0: (*Einschwingvorgang wird abgewartet*)
	BereitNachstePosition:= FALSE;
	IF ManuellOK THEN 
	timer_Einschwingen(IN:= TRUE, PT:= T#120S ); // der Timer wird gestartet, damit sich das Wägesystem einschwingen kann
	IF timer_Einschwingen.Q  THEN 
		timer_Einschwingen(IN :=FALSE); 
		ManuellOK := FALSE;
		state:=1;
	END_IF
	END_IF
	
1: (*Kalibrierungsdaten werden aufgenommen und über einen FIlter gemittelt*)
	
	timer_Messen(IN:= TRUE, PT:= T#120S); //120 Sekunden wird gemessen
	
	CASE  Kalibrierungsschritt OF
		1: 
			GesKaliGewicht := Kalibrierungsgewichte[1];
			//SM.Mitteilung  :='Bitte hängen';
		2:
			GesKaliGewicht := Kalibrierungsgewichte[2];
		3:
			GesKaliGewicht := Kalibrierungsgewichte[1] + Kalibrierungsgewichte [2];
		4:
			GesKaliGewicht := Kalibrierungsgewichte[2] + Kalibrierungsgewichte [3];
		5:
			GesKaliGewicht := Kalibrierungsgewichte[1] + Kalibrierungsgewichte [2]+ Kalibrierungsgewichte [3];
	END_CASE

	FilterIn :=Waage_Offset[WaagenNummer]/ GesKaliGewicht;
	Trigger(in:= FilterIn, PT:= T#1S, out=> , Trig=> );

	WertMitteln(IN:= Trigger.out, E:= Trigger.Trig, N:= 30, RST:= BereitNachstePosition, AVG=>k_werte[Kalibrierungsschritt] );	
	
	IF timer_Messen.Q THEN 
		state :=2;
		timer_Messen(IN:= FALSE);
	END_IF


2: (*Übertragung der k-Werte in das Kalibrierungs-Array*)

	Umrechnungsfaktoren[WaagenNummer,Kalibrierungsschritt]:= k_werte[Kalibrierungsschritt];

	state:= 3;

3:	

	BereitNachstePosition:= TRUE;
	Kalibrierungsschritt:= Kalibrierungsschritt + 1; //nächster Kalibrierungsschritt
	
	(*Falls eine Waage alle Kalibrierungsschritte durchlaufen hat wird die nächste Waage 
		kalibriert.*)
	IF Kalibrierungsschritt > 5 THEN 
		WaageKalibriert[WaagenNummer]:=TRUE;
		WaagenNummer := WaagenNummer +1 ;
		Kalibrierungsschritt := 1;
		state:= 0;
	END_IF
	
	(*Alle Waagen sind alle 5 Kalibrierungsschritte durchlaufen. Gewichtskalibrierung ist abgeschlossen
		state wird auf Null gesetzt.*)
	IF Kalibrierungsschritt > 5  AND WaagenNummer > 4 THEN 
			WaagenKalibrierungFertig:= TRUE; 
			state:= 0;
	END_IF

END_CASE

END_PROGRAM

// ---- POUs/Waagen/Lesen_Waagen.TcPOU
PROGRAM Lesen_Waagen
(* Dieses Program wird dazu verwendet den aktuellen Waagenwert(String) aus dem Zwischenspeicher (RxBuffer) 
	zu entnehmen. Nach der Verarbeitung im Funktionsbaustein werden alle Werte der Waage_X wieder sich
	zugewiesen und gespeichert. *)  

VAR
	fb_WaageAuslesen : ARRAY[1..6] OF FB_GewichtAuslesen;
	counter: INT;
	myOffset: REAL;
	
(*Variablen für Offset-Ermittlung *)
	Timer,Timer1: TON;
	Trigger:  ARRAY[1..4] OF SH_1;
	GetOffset:ARRAY[1..4] OF FT_AVG;;
	bOffset: 		BOOL := FALSE;
	//bGetOffset: 		BOOL;

	Offset_VD: BOOL;
END_VAR

VAR PERSISTENT 
	Offset_Tare: 	ARRAY[1..4] OF REAL; 
	Offset_Ventilator_AN: 		ARRAY[1..4] OF REAL; 
	Offset_Kaltemittel_g: 		ARRAY[1..4] OF REAL; 
	Offset_Kaltemittel_f: 		ARRAY[1..4] OF REAL; 
END_VAR

// 	Waagen 1..6 werden ausgelesen. 
FOR counter:= 1 TO 6 DO 
	fb_WaageAuslesen[counter](myWaage:= Waage[counter] , myBuffer:= RxBuffer[counter] , Waage=> Waage[counter] );
	Waage_roh[counter] := Waage[counter].Masse;
END_FOR

(*Offset für Ventilator wird immer berücksichtig, wenn VD an ist und keine Kalibrierung geschieht*)
IF DO_VD_Ventilator_ON= TRUE AND bGetOffset_Ventilator = FALSE THEN
	Offset_VD := TRUE;
	ELSE
	Offset_VD := FALSE;
END_IF


(*	Waagen 1..4 werden falls nötig mit einem OFFSET korrigiert. zB durch Laufen der Ventilatoren.
 OFFSET wird nicht berechnet, wenn der gerade ein Offset ermittelt wird*)

IF 	bTare = FALSE 	THEN
//AND bGetOffset_Ventilator = FALSE AND bGetOffset_Kaltemittel_g = FALSE AND	bGetOffset_Kaltemittel_l = FALSE THEN
FOR counter:= 1 TO 4 DO 
	Waage_Offset[counter] := OFFSET(
	X:= Waage[counter].Masse, 
	O1:= bOffset, 				//wird TRUE nach dem ersten TARE-Befehl. Waagen sind wieder bei '0g'
	O2:= Offset_VD, 
	O3:= VD_Kaltemittel_g, 
	O4:= VD_Kaltemittel_l, 
	D:=  FALSE, 
	Offset_1:= -Offset_Tare[counter],
	Offset_2:= -Offset_Ventilator_AN[counter],  
	Offset_3:= -Offset_Kaltemittel_g[counter], 
	Offset_4:= -Offset_Kaltemittel_f[counter], 
	default:= 10000);
END_FOR
END_IF



//CASE SM.Status OF
	
//Initialisieren: 

IF 	bTare 	OR bGetOffset_Ventilator 	 OR bGetOffset_Kaltemittel_g OR	bGetOffset_Kaltemittel_l THEN 
	bGetOffset_Abgeschlossen	:=FALSE;
	bTare_Abgeschlossen 		:=FALSE;
	bVentilator_Abgeschlossen	:=FALSE;
	Timer(IN:= TRUE, PT:=T#60S , Q=> , ET=> );
	bOffset 					:= TRUE;
	IF bTare THEN 
		bOffset:= FALSE;
	END_IF
END_IF

//Offset wird bestimmt für den Fall, dass die Waagen mit ca. 2000 g vorbelastet sind
	IF bTare THEN 
		FOR counter:= 1 TO 4 DO 
			Trigger[counter](in:= Waage[counter].Masse, PT:= T#1S, out=> , Trig=> );
			GetOffset[counter](IN:= Trigger[counter].out, E:= Trigger[counter].Trig, N:= 30, RST:= , AVG=>Offset_Tare[counter] );	
		END_FOR
			//bOffset:= TRUE;
	END_IF


//Offset wird bestimmt für den Fall, dass der VENTILATOR an ist
	IF bGetOffset_Ventilator THEN
		VD_Ventilator_ON:= TRUE;
		Timer1(IN:=TRUE, PT:= T#30S); 
		IF Timer1.Q THEN 
			FOR counter:= 1 TO 4 DO 
				Trigger[counter](in:= Waage_Offset[counter], PT:= T#1S, out=> , Trig=> );//Trigger[counter](in:= Waage[counter].Masse, PT:= T#1S, out=> , Trig=> );
				GetOffset[counter](IN:= Trigger[counter].out, E:= Trigger[counter].Trig, N:= 30, RST:= , AVG=>Offset_Ventilator_AN[counter] );	
			END_FOR
		//Timer1(IN:=FALSE);
		END_IF
	END_IF

//Offset wird bestimmt für den Fall, dass das KÄLTEMITTEL GASFÖRMIG ist
	IF bGetOffset_Kaltemittel_g THEN 
		FOR counter:= 1 TO 4 DO 
			Trigger[counter](in:= Waage[counter].Masse, PT:= T#1S, out=> , Trig=> );
			GetOffset[counter](IN:= Trigger[counter].out, E:= Trigger[counter].Trig, N:= 30, RST:= , AVG=>Offset_Kaltemittel_g[counter] );	
		END_FOR
	END_IF

//Offset wird bestimmt für den Fall, dass das KÄLTEMITTEL FLÜSSIG ist	
	IF bGetOffset_Kaltemittel_l THEN 	
		FOR counter:= 1 TO 4 DO 
			Trigger[counter](in:= Waage[counter].Masse, PT:= T#1S, out=> , Trig=> );
			GetOffset[counter](IN:= Trigger[counter].out, E:= Trigger[counter].Trig, N:= 30, RST:= , AVG=>Offset_Kaltemittel_f[counter] );	
		END_FOR
	END_IF

//Nachdem die Zeit abgelaufen ist, werden die BOOL-Variablen zurückgesetzt
	IF Timer.Q THEN
		
		//bOffset								:= TRUE;
		
		bGetOffset_Kaltemittel_g			:= FALSE; 
		bGetOffset_Kaltemittel_l 			:= FALSE;
	
		IF bGetOffset_Ventilator = TRUE THEN
			VD_Ventilator_ON	:=		FALSE;
			bGetOffset_Ventilator:=		FALSE;
			bVentilator_Abgeschlossen:=	TRUE;
		END_IF
	
		IF bTare= TRUE THEN 
			bOffset						:= TRUE; //ermittelter Offset wird wieder vom Rohwert abgezogen
			bGetOffset_Abgeschlossen	:= TRUE;	
			bTare    					:= FALSE;
		END_IF
		Timer(IN:= FALSE);	
		Timer1(IN:=FALSE);
	END_IF
	
//END_CASE

END_PROGRAM

// ---- POUs/Funktionen/FB_GewichtAuslesen.TcPOU
FUNCTION_BLOCK FB_GewichtAuslesen

VAR_INPUT
	myWaage: WAAGE_VAR;		// Eine Inputvariable myWaage wird als WAAGE_VAR deklariert.
END_VAR

VAR_IN_OUT
	myBuffer:ComBuffer;		// Ein Zwischenspeicher wird deklariert. Buffer immer als VAR_IN_OUT deklarieren
END_VAR

VAR

(*Es folgen Variabeln die der FB ReceiveString benötigt*)
	ReceiveString_Buffer:	ReceiveString;
	tTimeout: 				TIME;
	bReset: 				BOOL;
	bStringReceived:		BOOL;
	bbusy:					BOOL;
	bRxTimeout: 			BOOL;
	eError: 				ComError_t;
	stLastStringReceived: 	STRING;
	stReceivedString: 		STRING;


	Var1: INT;				//1.Stringlänge
	Var2: INT;				//2.Stringlänge
	Var3: INT;				//3.Stringlänge
	MyString: STRING(80);	//
	Position_g: INT;		// Position des Grammzeichens 'g'. Ausgabe von Waage nur bei stabilen Werten
END_VAR
VAR_OUTPUT
	Waage: WAAGE_VAR (*:= myWaage*) ;  
END_VAR

//Empfange Datenstring aus dem Datenpuffer RxBuffer der jeweiligen Waage
ReceiveString_Buffer(
	Prefix:= '', 
	Suffix:= '$R$N', 
	Timeout:=tTimeout , 
	Reset:=bReset , 
	StringReceived=>bStringReceived , 
	Busy=>bbusy , 
	Error=>eError, 
	RxTimeout=> bRxTimeout ,
	ReceivedString:= stReceivedString, 
	RXbuffer:= myBuffer);

//Übergabe des empfangenen Strings an MyString und Längenabfrage
MyString:= stReceivedString;
Var1:= LEN (MyString);


//Löschen von $R$N aus MyString und Längenabfrage
MyString := DELETE (MyString,4,16); 
Var2:= LEN (MyString);


//Löschen der Leerzeichen aus MyString und Längenabfrage
WHILE FIND(MyString,' ') <> 0 DO
	MyString:=DELETE (MyString,1,FIND(MyString,' '));
END_WHILE
Var3:= LEN (MyString);


(*Überprüfen ob ein stabiler Messwert an der Waage anliegt
	Falls 'g' in MySting vorhanden 		-> Boolvariable bStabilerWert TRUE
	Falls kein 'g' in MyString vorhanden-> Boolvariable bStabilerWert FALSE	*)
Position_g := FIND(MyString,'g');
CASE Position_g OF
		0: myWaage.bStabilerWert := FALSE;
	ELSE
		myWaage.bStabilerWert := TRUE;
END_CASE


// Übergabe von MyString in Realvariable MyReal

myWaage.Masse:=STRING_TO_REAL(MyString);

Waage:= myWaage;

END_FUNCTION_BLOCK

// ---- POUs/Modbus/Lesen_Modbus.TcPOU
PROGRAM Lesen_Modbus
(*In diesem Programm werden alle Modbus-Daten umgerechnet. *)

VAR
	Auslesen0, Auslesen1, Auslesen2, Auslesen3, Auslesen4, Auslesen5, Auslesen6, Auslesen7, Auslesen8 : FB_fpconverter;
	
	EV1 : FB_EVconverter;		//Funktionsbaustein zur Auswertung eines Expansionsventiles
	EV2 : FB_EVconverter;		//Funktionsbaustein zur Auswertung eines Expansionsventiles
	FP_Umrechnen : FB_fpconverter;	//Funktionsbaustein zur Umrechnung von FLOAT->REAL
END_VAR

(*Auslesen der Druckdaten der 8 Drucksensoren im Kältekreis*)
Auslesen1(myPT:= PT_KP_in, 	PT=> PT_KP_in);
Auslesen2(myPT:= PT_KP_out, PT=> PT_KP_out);
Auslesen3(myPT:= PT_VF_in,	PT=> PT_VF_in);
Auslesen4(myPT:= PT_VF_out, PT=>PT_VF_out );
Auslesen5(myPT:= PT_vor_EV, PT=>PT_vor_EV );
Auslesen6(myPT:= PT_vor_EV_rev, PT=>PT_vor_EV_rev );
Auslesen7(myPT:= PT_VD_in,  PT=> PT_VD_in);
Auslesen8(myPT:= PT_VD_out, PT=> PT_VD_out);

(*Deklarierung der ModbusData_Startfelder der Slaves Modbus. Hier schreibt der ModbusRTU die empfangenden Daten hinein
	Startfeld entspricht zur Übersicht der Modbus-Adresse. *)
PT_KP_in.Startfeld_ModbusData		:= 4;
PT_KP_out.Startfeld_ModbusData		:= 5;
PT_VF_in.Startfeld_ModbusData		:= 6;
PT_VF_out.Startfeld_ModbusData		:= 7;
PT_vor_EV.Startfeld_ModbusData		:= 8;
PT_vor_EV_rev.Startfeld_ModbusData 	:= 9;
PT_VD_in.Startfeld_ModbusData		:= 10;
PT_VD_out.Startfeld_ModbusData		:= 11;

(*Expansionsventile werden ausgelesen und umgerechnet*)
EV1(inEV:=EV , outEV=> EV);
EV2(inEV:=EV_rev, outEV=> EV_rev);

(*Daten vom Massestromsensoren werden umgerechnet. FLOAT-Werte werden in REAL umgerechnet*)
MSS.rFliessgeschwindigkeit	:= FloatPointDW_TO_REAL(MSS.Data[1]);
MSS.rVolumenstrom			:= FloatPointDW_TO_REAL(MSS.Data[2]);
MSS.rMassenstrom			:= FloatPointDW_TO_REAL(MSS.Data[3])*1000; // wird nun angezeigt in [g/s]
MSS.rTemp					:= K_TO_C(FloatPointDW_TO_REAL(MSS.Data[4]));
MSS.rDichte					:= FloatPointDW_TO_REAL(MSS.Data[5]);

END_PROGRAM

// ---- POUs/Funktionen/FB_fpconverter.TcPOU
FUNCTION_BLOCK FB_fpconverter 
(* Dieser FB dient zur Umrechnung der DATABYTEs in einen REAL-Wert.
	Je nach ausgeführtem Modbus-Befehl(nur Druck oder Temperatur, oder beides) werden
	unterschiedlich viele DATABYTEs von dem Drucksensor geschickt. 
	Die Boolvariablen zur Druck- und Temperaturabfrage müssen durch den User gesetzt werden.
	Der FB gibt den Druck und die Temperatur in REAL an die STRUCT Drucksensor zurück.*)

VAR_INPUT
	myPT : Drucksensor;
END_VAR
VAR
	myString_druck: STRING(32);
	myString_temp: STRING(32);
END_VAR

VAR_OUTPUT
		PT: Drucksensor;
END_VAR

//Umrechnung der BYTEs in Binär-STRINGs und zusammensetzen der 4 DATA-BYTEs zu einem 32 bit STRING
myPT.Data[0]:= ModbusRTU_COM.modbusData_PT[myPT.Startfeld_ModbusData];

	IF myPT.bDruckabfrage THEN
		myString_druck:=DWORD_TO_BINSTRING(ModbusRTU_COM.modbusData_PT[myPT.Startfeld_ModbusData]);
		myPT.rDruck:=BINSTRING_TO_REAL(myString_druck); 		// tatsächlicher Druck in Bar
	ELSE
		myPT.rDruck:=0;	
	END_IF
	
	
(*Umrechnung für Temperatur, falls bTemperaturabfrage gleich TRUE *)	
	IF myPT.bTemperaturabfrage  THEN
		myString_druck:=DWORD_TO_BINSTRING(ModbusRTU_COM.modbusData_PT[myPT.Startfeld_ModbusData]);
		myPT.rTemp:= BINSTRING_TO_REAL(myBinString:= myString_temp); 		//Umrechnung nach IEEE 754 von 32 bit floating point zur REAL-Variable 
	ELSE
		myPT.rTemp:= 0;
	END_IF

PT := myPT;

END_FUNCTION_BLOCK

// ---- POUs/Modbus/ModbusRTU_COM.TcPOU
PROGRAM ModbusRTU_COM

(*Dieses Programm komuniziert über einen MODBUS-RTU mit den installieren Drucksensoren(PT),
den E-Ventilen und dem Massenstromsensor im Kältekreislauf. Die Senoren/Aktoren besitzen eine 
eindeutige Adresse. Über die Adressen werden sie vom MASTER(Pc) angesprochen und führen die
verlange Funktion durch.

Dieses Programm ist erst nach Initialierung, sprich Zuweisung der Adressen, zu verwenden.
Wenn mehrere Sensoren/Aktoren die gleiche Adresse haben, kommt es zu Fehlern in der Kommunikation.
Die Kommunikation verläuft in einer CASE-Struktur.*)

VAR
(*
_________________________________________________________	
Drucksensoren	|	Position im RI	|	Modbus-Adresse
PT_KP_in		|	1				|	4
PT_KP_out		|	2				|	5
PT_VF_in		|	2‘ 				|	6
PT_VF_out		|	3‘ 				|	7
PT_vor_EV 		|	3 (innerhalb KK)|	8 
PT_vor_EV_rev 	|	3 (außerhalb KK)|	9
PT_VD_in		|	4				|	10
PT_VD_out		|	1‘ 				|	11
__________________________________________________________
Massenstromsensor
MSS 1			|	3				|	12 
*)
	
	state: INT;

(*Variablen für die Modbus-Befehle*)
	 ModbusAdresse: 	BYTE := 3;
	 modbusData_PT: 	ARRAY[0..12] OF DWORD;		//hier werden die Daten von den Drucksensoren gespeichert
	 
(*Abfrageregister vom MassenstromSensor*)
	AbfrageRegs_MSS:ARRAY[1..5] OF INT := [30000,30002,30004,30006,30008]; 	

(*Abfrageregister vom MassenstromSensor*)
	AbfrageRegs_PT:WORD := 2; 	
	LaengeRegs: BYTE:= 2;
	
(*Variablen für Error- und Successzähler der Modbus-Komunikation *)
	FtrigBusy:			F_TRIG;
	LastErrorstate: 	INT;
	LastModbusError: 	ST_ModbusErrorDiagnostics;
	CounterError: 		DINT;
	CounterSuccess: 	DINT;
	counter: 			INT := 1;
	Teststring: T_MaxString;
END_VAR

(*Falls ein Slave konfiguriert werden soll bConfigPT auf TRUE setzen*)
		
IF 	bConfigPT THEN 
	Status_Modbus := ConfigPT;
ELSE 
	Status_Modbus := Aktiv;
END_IF


CASE Status_Modbus OF
	
Aktiv: 

CASE state OF

0: (*Initialisierung von Modbus und Durchzählen der Modbus-Adressen*)
		MODBUS.myModbus.ReadRegs(Execute:= FALSE);
		MODBUS.myModbus.WriteRegs(Execute:= FALSE);

		
		ModbusAdresse := ModbusAdresse + 1;		//Laufvariable für die ModbusAdressen der Slaves. Zunächst nur Drucksensoren.
		IF ModbusAdresse >= 13 THEN				//alle PTs und der Massenstromsensor werden ausgelesen
			ModbusAdresse := 4;
		END_IF
		
		
		state := state + 1;


1:	(* Lese Keller-Registers aus*)	
     
	IF ModbusAdresse<=11 AND ModbusAdresse>=4 THEN 
	 MODBUS.myModbus.ReadRegs (* Reads data from a connected slave. *)
 		(
 		 UnitID:= ModbusAdresse,
 		 Quantity:= LaengeRegs,								//zwei Register werden ausgelesen
 		 MBAddr:= AbfrageRegs_PT,								//P1 wird bei Adresse 2 ausgelesen, TOB1 bei Adresse 8
 		 cbLength:= SIZEOF(modbusData_PT[ModbusAdresse]),		
 		 pMemoryAddr:= ADR(modbusData_PT[ModbusAdresse]),		//Empfangene Daten werden in DWORD in modbusData geschrieben.
  		Execute:= TRUE,
  		Timeout:= modbusTimeout,
  		Busy => Modbus.isModbusBusy,
  		Error => isModbusError,
  		ErrorId => modbusErrorId
  		(* cbRead parameter *));
		
  		IF NOT isModbusBusy THEN
				MODBUS.myModbus.ReadRegs(Execute:= FALSE);
			IF MODBUS.myModbus.Error THEN
				state := 0;
			ELSE
				state := state + 1;
			END_IF
		END_IF
		ELSE 
		state := state + 1;
	END_IF
	
	
	
2:	(* Lese Massenstromsensor-Registers aus*)		
	(*	Folgende Messdaten werden ausgelesen:
			
				   Messgröße		|	Einheit	|	Register-Adressen
				____________________|___________|_____________________   
				1) Fließgeschw.     |	[m/s]	|	30000-2 Regs
				2) Volumenstrom		|	[m³/s]	|	30002-2 Regs
				3) Massenstrom		|	[kg/s]	|	30004-2 Regs
				4) Temperatur		|	[K]		|	30006-2 Regs
				5) Dichte			|	[kg/m³]	|	30008-2 Regs			->ingesamt 10 Regs
		*) 
	IF ModbusAdresse=12 THEN	
		myModbus.ReadInputRegs(
		UnitID:= 12,
 		Quantity:= 2,							
 		MBAddr:= INT_TO_WORD(AbfrageRegs_MSS[counter]),								
 		cbLength:= SIZEOF(MSS.Data[counter]),		
 		pMemoryAddr:= ADR(MSS.Data[counter]),	 
  		Execute:= TRUE,
  		Timeout:= modbusTimeout,
  		Busy => isModbusBusy,
  		Error => isModbusError,
  		ErrorId => modbusErrorId
  		(*cbRead parameter)*));
	
			IF isModbusBusy = FALSE AND counter<=5 THEN
				myModbus.ReadInputRegs(Execute:= FALSE);
				counter:= counter +1;
			END_IF	
			
			IF isModbusBusy = FALSE AND counter>5 THEN
				myModbus.ReadInputRegs(Execute:= FALSE);
				counter:=1;
				state:= 0;
			END_IF	
	ELSE 
		state:= 0;
	END_IF	
END_CASE	

ConfigPT:
	
	ConfigDrucksensor(); 		//Programm für Konfigurierung von Keller-Drucksensoren

END_CASE 

// Zählen der erfolgreichen und fehlerhaften Komunikationsschritte 
FtrigBusy(CLK:=myModbus.BUSY );
IF FtrigBusy.Q THEN
	IF MODBUS.myModbus.Error THEN
		LastModbusError := MODBUS.myModbus.ErrorDiagnostics;
		LastErrorstate := state;
		CounterError := CounterError + 1;
	ELSE
		CounterSuccess := CounterSuccess + 1;
	END_IF
END_IF

END_PROGRAM

// ---- POUs/Modbus/ConfigDrucksensor.TcPOU
PROGRAM ConfigDrucksensor
VAR
	state : INT := 1;
	
	(*Daten für die Konfiguration vom Keller-Drucksensor*)	
	UART_akt: 				WORD;
	UARTsettings_akt:		ARRAY[0..1]OF BYTE;
	UARTsettings_neu: 		ARRAY[0..1]OF BYTE  ;//:= [48,0];
	wUARTsettings_neu:		WORD := 0;//:= 112;
	sUARTsettings_neu: 		STRING;
	ModbusRegister:   		Word := 17;
	RegisterLange: 			BYTE := 1;
	ModbusAddress_alt: 		WORD {1..250}:= 1;			//alte Modbusadresse des Slaves. Anfangs gleich der Auslieferungsadresse
	ModbusAddress_neu: 		WORD {3..12} := 11;				//neue Modbusadresse des Slaves. 
	ModbusDataTest: 		DWORD;
	Teststring: 			STRING;
END_VAR

(*Keller-Slaves Konfiguration*)

Teststring:= DWORD_TO_BINSTR(ModbusDataTest,32);

CASE MODBUS.Status_Modbus OF

ConfigPT:

CASE state OF
1:   (* Write Register, write new address to Slave *)	
		IF bConfigPT_setadresse THEN
	 	MODBUS.myModbus.WriteSingleRegister (* writes data to a connected slave. *)
 		(
 		 UnitID:= WORD_TO_BYTE(ModbusAddress_alt),
 		 Quantity:= 1,
 		 MBAddr:= 525,							//Keller: DEV_ADDR 0x020D= DECx525
 		 cbLength:= SIZEOF(ModbusAddress_neu),
 		 pMemoryAddr:= ADR(ModbusAddress_neu),
  		Execute:= TRUE,
  		Timeout:= modbusTimeout,
  		Busy => isModbusBusy,
  		Error => isModbusError,
  		ErrorId => modbusErrorId
  		(* cbRead parameter *));
		
  		IF NOT isModbusBusy THEN
				MODBUS.myModbus.WriteSingleRegister(Execute:= FALSE);
			IF MODBUS.myModbus.Error THEN
				state := 2;
			ELSE
				state := 2;	
			END_IF
		END_IF
		ELSE
			state:= 2;
		END_IF
	
2: 	(* TEST-READ Regs from connected Slave *)

		 MODBUS.myModbus.ReadRegs 
 		(
 		 UnitID:= WORD_TO_BYTE(ModbusAddress_neu),
 		 Quantity:= RegisterLange,						//2 Regs für den Druck P1 oder Temperatur TOB1
 		 MBAddr:= ModbusRegister,						//DECx02 Reg-Adresse für P1, DECx08 Reg-Adresse für TOB1
 		 cbLength:= SIZEOF(ModbusDataTest),
 		 pMemoryAddr:= ADR(ModbusDataTest),
  		Execute:= TRUE,
  		Timeout:= modbusTimeout,
  		Busy => isModbusBusy,
  		Error => isModbusError,
  		ErrorId => modbusErrorId
  		(* cbRead parameter *));
		
  		IF NOT isModbusBusy THEN
				MODBUS.myModbus.ReadRegs(Execute:= FALSE);
			IF myModbus.Error THEN
				state := 2;
			ELSE
				state := 1;	
			END_IF
		END_IF
		
3: (* Write Register, write new UART-settings to Slave *)
	IF bConfigPT_setUART THEN
	 	MODBUS.myModbus.WriteSingleRegister (* writes data to a connected slave. *)
 		(
 		 UnitID:= WORD_TO_BYTE(ModbusAddress_neu),
 		 Quantity:= 1,
 		 MBAddr:= 512,							//Keller: DEV_ADDR 0x020D= DECx525
 		 cbLength:= SIZEOF(wUARTsettings_neu),
 		 pMemoryAddr:= ADR(wUARTsettings_neu),
  		Execute:= TRUE,
  		Timeout:= modbusTimeout,
  		Busy => isModbusBusy,
  		Error => isModbusError,
  		ErrorId => modbusErrorId
  		(* cbRead parameter *));
		
		sUARTsettings_neu:= CONCAT(BYTE_TO_STRING(UARTsettings_neu[1]), BYTE_TO_STRING(UARTsettings_neu[0]));
  		IF NOT isModbusBusy THEN
				MODBUS.myModbus.WriteSingleRegister(Execute:= FALSE);
			IF MODBUS.myModbus.Error THEN
				state := 1;
			ELSE
				state := 4;	
			END_IF
		END_IF
	ELSE
		state:= 4;
  	END_IF

4: (* Read UART-Register from Slave *)

	 	MODBUS.myModbus.ReadRegs
 		(
 		 UnitID:= WORD_TO_BYTE(ModbusAddress_neu),
 		 Quantity:= 1,
 		 MBAddr:= 512,							//Keller: DEV_ADDR 0x020D= DECx525
 		 cbLength:= SIZEOF(UARTsettings_akt),
 		 pMemoryAddr:= ADR(UARTsettings_akt),
  		Execute:= TRUE,
  		Timeout:= modbusTimeout,
  		Busy => isModbusBusy,
  		Error => isModbusError,
  		ErrorId => modbusErrorId
  		(* cbRead parameter *));
		
		//Ändert die Byte-Reihenfolge und konvertiert sie in ein WORT
		UART_akt:= WORD_OF_BYTE(UARTsettings_akt[1], UARTsettings_akt[0]);
		
		
  		IF NOT isModbusBusy THEN
				MODBUS.myModbus.ReadRegs(Execute:= FALSE);
			IF MODBUS.myModbus.Error THEN
				state := 3;
			ELSE
				state := 4;	
			END_IF
		END_IF
		
END_CASE

END_CASE

END_PROGRAM

// ---- POUs/Funktionen/DWORD_TO_BINSTRING.TcPOU
FUNCTION DWORD_TO_BINSTRING : STRING(32)
VAR_INPUT
	myDWORD:DWORD;		//DWORD aus der Klemme/Modbusarray
END_VAR
VAR
		b3: BYTE; 
		b2: BYTE;
		b1: BYTE;
		b0: BYTE;
		s3: STRING(8);
		s2: STRING(8);
		s1: STRING(8);
		s0: STRING(8);
END_VAR

(*da Twincat mit LIL-Endian arbeitet und die Kellersensoren mit BIG-Endian,
 müssen die Bytes paarweise vertauscht werden*)

//Zerteilen des DWORDs in die 4 Bytes
b3:= BYTE_OF_DWORD(myDWORD, 1);
b2:= BYTE_OF_DWORD(myDWORD, 0);
b1:= BYTE_OF_DWORD(myDWORD, 3);
b0:= BYTE_OF_DWORD(myDWORD, 2);

//Umrechnung der BYTES in Binärestrings mit der Länge 8 bits
s3:= BYTE_TO_BINSTR(b3,8);
s2:= BYTE_TO_BINSTR(b2,8);
s1:= BYTE_TO_BINSTR(b1,8);
s0:= BYTE_TO_BINSTR(b0,8);

//Zusammenfügen der vier Binärstrings zu einem 32 bit String
DWORD_TO_BINSTRING := CONCAT(CONCAT(s3,s2), CONCAT(s1,s0));

END_FUNCTION

// ---- POUs/Funktionen/BINSTRING_TO_REAL.TcPOU
FUNCTION BINSTRING_TO_REAL : REAL
	(*Ein 32 bit Binärstring wird in einen REAL-Wert umgerechnet*)
VAR_INPUT
	myBinString : STRING(32);
END_VAR
VAR
	stSign: STRING(1);
	rSign: 	REAL;
	Sign: 	BOOL;
	
	stExponent: STRING(8);
	Exponent: 	UINT;
	
	stMantis: 	STRING(23);
	Mantis: 	DWORD;

END_VAR

	
	stSign		:= LEFT(myBinString,1);
	Sign		:= STRING_TO_BOOL(stSign);
	rSign		:= STRING_TO_REAL(stSign);

	stExponent	:= RIGHT(LEFT(myBinString,9),8);	
	Exponent	:= BYTE_TO_UINT(BIN_TO_BYTE(stExponent));

	stMantis	:= RIGHT(myBinString,23);
	Mantis		:= BIN_TO_DWORD(stMantis);

	BINSTRING_TO_REAL:= FPU.ComposeRealRaw(bS:=Sign , uiE:= Exponent, udiM:= Mantis ); // Ergebnis in REAL

END_FUNCTION

// ---- POUs/Funktionen/FB_EVconverter.TcPOU
FUNCTION_BLOCK FB_EVconverter
VAR_INPUT
	inEV : ExpansionsVentil;
END_VAR
VAR
END_VAR

VAR_OUTPUT
	 outEV : ExpansionsVentil;
END_VAR

	inEV.IstDruck :=	 	INT_TO_REAL(WORD_TO_INT(inEV.modbusData[1]))/10;
	inEV.IstTemp:=	 		INT_TO_REAL(WORD_TO_INT(inEV.modbusData[2]))/10;
	inEV.SaugTemp:= 		INT_TO_REAL(WORD_TO_INT(inEV.modbusData[3]))/10;
	inEV.VerdampfTemp:= 	INT_TO_REAL(WORD_TO_INT(inEV.modbusData[4]))/10;
	inEV.VerdampfDruck:= 	INT_TO_REAL(WORD_TO_INT(inEV.modbusData[5]))/10;
	inEV.UberhitzungTemp:= 	INT_TO_REAL(WORD_TO_INT(inEV.modbusData[6]))/10;
	inEV.VentilOffnung:= 	INT_TO_REAL(WORD_TO_INT(inEV.modbusData[7]))/10;
	inEV.RegelSollwert:= 	INT_TO_REAL(WORD_TO_INT(inEV.modbusData[8]))/10;
	inEV.Ventilposition:= 	INT_TO_REAL(WORD_TO_INT(inEV.modbusData[9]));
	inEV.AktKuhlleistung:= 	INT_TO_REAL(WORD_TO_INT(inEV.modbusData[10]));
	
	inEV.LOP := inEV.modbusDataCoils[1];
	inEV.MOP := inEV.modbusDataCoils[2];
	inEV.LowSH:= inEV.modbusDataCoils[3];
	inEV.HiTcond:= inEV.modbusDataCoils[4];
	
	outEV:= inEV;

END_FUNCTION_BLOCK

// ---- POUs/Funktionen/FloatPointDW_TO_REAL.TcPOU
FUNCTION FloatPointDW_TO_REAL : REAL
(*Diese Funktions rechnet 32 bit FLOAT-Werte in einen REAL-Wert um und gibt diesen wieder aus.*)
VAR_INPUT
	in : DWORD;
END_VAR
VAR
	BinString : STRING;
END_VAR

(*DWORD wird in einen Binären 32bit String umgewandelt*) 
BinString:= DWORD_TO_BINSTR(in,32);
 
 (*Binärstring wird in eine REAL Variable umgerechnet*)
 FloatPointDW_TO_REAL:= BINSTRING_TO_REAL(myBinString:= BinString);

END_FUNCTION

// ---- POUs/Modbus/ModbusRTU_EL.TcPOU
PROGRAM ModbusRTU_EL
VAR
(*Modbus für Klemme EL6021 wird deklariert*)
	ModbusEL6021:		ModbusRtuMaster_KL6x22B;	
	modbusTimeout_EL:	TIME := T#300MS;
	isModbusBusy_EL:	BOOL;
	isModbusError_EL:	BOOL;
	modbusErrorId_EL:	MODBUS_ERRORS;
	
(*Hilfsvariablen für Modbus	

Sensor/Aktor	|	Position		|	Modbus-Adresse
________________|___________________|____________________
EV				|	3				|	2
EV_rev			|	3				|	3	
*)
	//modbusData_EV: 	ARRAY[1..10] OF INT;		//hier werden die Daten vom EV gespeichert
	EV_Adresse : BYTE := 2;				//ModbusAdresse vom Expansionsventil	
	EV_rev_Adresse : BYTE := 3;			//ModbusAdresse vom Abtau-Expansionsventil
	state: 			INT := 0;
	counter: 		INT := 1;
	
	AbfrageRegs: ARRAY [1..10] OF WORD := [0,1,4,5,6,9,16,20,131,134]; 	//Modbus-Register-Adressen. Das sind alle Werte die vom EV abgefragt werden
	AbfrageCoils: ARRAY [1..4] OF WORD := [49,50,51,52];					//Modbus-Coil-Adressen.
	
(*Variablen für Error- und Successzähler der Modbus-Komunikation *)
	FtrigBusy:			F_TRIG;
	LastErrorstate: 	INT;
	LastModbusError: 	ST_ModbusErrorDiagnostics;
	CounterError: 		DINT;
	CounterSuccess: 	DINT;

	TestMSS: ARRAY [0..10] OF DWORD;
END_VAR


CASE state OF

0: (*Initialisierung von Modbus*)
	
		ModbusEL6021.ReadInputRegs(Execute:= FALSE);
		ModbusEL6021.ReadCoils(Execute:= FALSE);
		ModbusEL6021.WriteSingleRegister(Execute:= FALSE);

		state :=1;
		
1: (*Liest Register von EV aus*)
 	
		ModbusEL6021.ReadInputRegs(
		UnitID:= EV_Adresse,
 		Quantity:= 1,								
 		MBAddr:= AbfrageRegs[counter],								
 		cbLength:= SIZEOF(EV.modbusData[counter]),//EV.modbusData[counter]),		
 		pMemoryAddr:= ADR(EV.modbusData[counter]),//EV.modbusData[counter]),		//Daten werden in für EV DATA-ARRAY geschrieben
  		Execute:= TRUE,
  		Timeout:= modbusTimeout_EL,
  		Busy => isModbusBusy_EL,
  		Error => isModbusError_EL,
  		ErrorId => modbusErrorId_EL
  		(*cbRead parameter)*));

		IF NOT isModbusBusy_EL THEN
				ModbusEL6021.ReadInputRegs(Execute:= FALSE);
			IF MODBUS.myModbus.Error THEN
				state := 0;
				ELSE
				counter := counter + 1;	
					IF counter > 10 THEN		//alle deklarierten Modbus-Register werden ausgelesen
					counter := 1;
					state:= 2;
					END_IF
			END_IF
		END_IF
		


	
2: (*Liest Coils von EV aus*)
		ModbusEL6021.ReadCoils(
		UnitID:= EV_Adresse,
 		Quantity:= 1,								
 		MBAddr:= AbfrageCoils[counter],								
 		cbLength:= SIZEOF(EV.modbusDataCoils[counter]),		
 		pMemoryAddr:= ADR(EV.modbusDataCoils[counter]),		//Daten werden in für EV DATA-ARRAY geschrieben
  		Execute:= TRUE,
  		Timeout:= modbusTimeout_EL,
  		Busy => isModbusBusy_EL,
  		Error => isModbusError_EL,
  		ErrorId => modbusErrorId_EL
  		(*cbRead parameter)*));
		
		IF NOT isModbusBusy_EL THEN
				ModbusEL6021.ReadCoils(Execute:= FALSE);
			IF ModbusEL6021.Error THEN
				state := 0;
			ELSE
				counter:= counter+1;
				IF counter > 4 THEN		//alle deklarierten Modbus-Register werden ausgelesen
					counter := 1;
					state:= 3;
				END_IF
			END_IF
		END_IF
		
3: (*Schreibt Akt_Kühlleistung Coil auf die Expansionsventile*)
IF EV.SetKuhlleistung THEN 	
	ModbusEL6021.WriteSingleRegister(
		UnitID:= EV_Adresse,
 		Quantity:= 1,								
 		MBAddr:= 134,								
 		cbLength:= SIZEOF(EV.SollKuhlleistung),		
 		pMemoryAddr:= ADR(EV.SollKuhlleistung),		//Daten werden in für EV DATA-ARRAY geschrieben
  		Execute:= TRUE,
  		Timeout:= modbusTimeout_EL,
  		Busy => isModbusBusy_EL,
  		Error => isModbusError_EL,
  		ErrorId => modbusErrorId_EL
  		(*cbRead parameter)*));

		IF NOT isModbusBusy_EL THEN
				ModbusEL6021.WriteSingleRegister(Execute:= FALSE);
				EV.SetKuhlleistung := FALSE;
			IF ModbusEL6021.Error THEN
				state := 0;
			ELSE
				state:= 4;
			END_IF
		END_IF
	ELSE 
		state:= 4;
END_IF
	
4: (*Liest Register von EV_rev aus*)
 	
		ModbusEL6021.ReadInputRegs(
		UnitID:= EV_rev_Adresse,
 		Quantity:= 1,								
 		MBAddr:= AbfrageRegs[counter],								
 		cbLength:= SIZEOF(EV_rev.modbusData[counter]),//EV.modbusData[counter]),		
 		pMemoryAddr:= ADR(EV_rev.modbusData[counter]),//EV.modbusData[counter]),		//Daten werden in für EV DATA-ARRAY geschrieben
  		Execute:= TRUE,
  		Timeout:= modbusTimeout_EL,
  		Busy => isModbusBusy_EL,
  		Error => isModbusError_EL,
  		ErrorId => modbusErrorId_EL
  		(*cbRead parameter)*));

		IF NOT isModbusBusy_EL THEN
				ModbusEL6021.ReadInputRegs(Execute:= FALSE);
			IF MODBUS.myModbus.Error THEN
				state := 0;
				ELSE
				counter := counter + 1;	
					IF counter > 10 THEN		//alle deklarierten Modbus-Register werden ausgelesen
					counter := 1;
					state:= 5;
					END_IF
			END_IF
		END_IF
		


	
5: (*Liest Coils von EV_rev aus*)
		

		ModbusEL6021.ReadCoils(
		UnitID:= EV_rev_Adresse,
 		Quantity:= 1,								
 		MBAddr:= AbfrageCoils[counter],								
 		cbLength:= SIZEOF(EV_rev.modbusDataCoils[counter]),		
 		pMemoryAddr:= ADR(EV_rev.modbusDataCoils[counter]),		//Daten werden in für EV DATA-ARRAY geschrieben
  		Execute:= TRUE,
  		Timeout:= modbusTimeout_EL,
  		Busy => isModbusBusy_EL,
  		Error => isModbusError_EL,
  		ErrorId => modbusErrorId_EL
  		(*cbRead parameter)*));

		IF NOT isModbusBusy_EL THEN
				ModbusEL6021.ReadCoils(Execute:= FALSE);
			IF ModbusEL6021.Error THEN
				state := 0;
			ELSE
				counter:= counter+1;
				IF counter > 4 THEN		//alle deklarierten Modbus-Register werden ausgelesen
					counter := 1;
					state:= 6;
				END_IF
			END_IF

		END_IF

6: (*Schreibt Akt_Kühlleistung Coil auf die Expansionsventile*)

IF EV_rev.SetKuhlleistung THEN 	
	ModbusEL6021.WriteSingleRegister(
		UnitID:= EV_rev_Adresse,
 		Quantity:= 1,								
 		MBAddr:= 134,								
 		cbLength:= SIZEOF(EV_rev.SollKuhlleistung),		
 		pMemoryAddr:= ADR(EV_rev.SollKuhlleistung),		//Daten werden in für EV DATA-ARRAY geschrieben
  		Execute:= TRUE,
  		Timeout:= modbusTimeout_EL,
  		Busy => isModbusBusy_EL,
  		Error => isModbusError_EL,
  		ErrorId => modbusErrorId_EL
  		(*cbRead parameter)*));

		IF NOT isModbusBusy_EL THEN
				ModbusEL6021.WriteSingleRegister(Execute:= FALSE);
				EV_rev.SetKuhlleistung := FALSE;
			IF ModbusEL6021.Error THEN
				state := 0;
			ELSE
				state:= 0;
			END_IF
		END_IF
	ELSE 
		state:= 0;
END_IF	
END_CASE

FtrigBusy(CLK:=ModbusEL6021.BUSY );
(*zählt fehlgeschlagene und erfolgreiche Komunikationsschritte*)
IF FtrigBusy.Q THEN
	IF ModbusEL6021.Error THEN
		LastModbusError := ModbusEL6021.ErrorDiagnostics;
		LastErrorstate := state;
		CounterError := CounterError + 1;
	ELSE
		CounterSuccess := CounterSuccess + 1;
	END_IF
END_IF

END_PROGRAM

// ---- POUs/Vereisung.TcPOU
PROGRAM Vereisung
(*Ablaufprogram für die Vereisung des Verdampfers. Beim ABBRUCH des Vorgangs bzw. ABSCHALTEN wird ein PumpDown vollzogen.  *)
VAR

END_VAR

(*Starte Timer zur Vereisung*)	
	IF NOT TimerVereisung.IN THEN
	TimerVereisung(IN:= TRUE, PT:= Vereisungszeit);
	END_IF
 		
	IF SM.bKuehlen THEN 
		fb_Schuetzstellung(myStatus := KuehlenOben);
	END_IF
	
(*Abtauung wird begonnen wenn Zeit des Timers abgelaufen ist*)
	IF TimerVereisung.Q THEN
		TimerVereisung.IN := FALSE;			//Reset vom Vereisungstimer
		Mitteilung:= 'Die Vereisungszeit ist abgeschlossen';
		
		(*Nach der Vereisung wird ein PumpDown durchgeführt*)
		SM.bPumpDown := TRUE; 
		
		(* Status-Maschine Bool-variablen werden auf TRUE bzw. FALSE gesetzt*)
		SM.bKuehlen := FALSE;	

		IF AutomatikZyklusEin THEN 
				bAbtauen := TRUE; 
				bPumpDown_revAbgeschlossen := FALSE;		//damit wieder ein PUMPDOWN rev im nächsten Zyklus durchgeführt werden kann
				CASE  AutomatikAbtauModus OF 
						NichtAusgewahlt: 
							Mitteilung := 'Kein Automatik-Abtaumodus ausgewählt!';
						Abtauen_elektrisch:
							bAbtauen_elektrisch := TRUE;
						Abtauen_Heissgas_oben:
							bAbtauen_Heissgas_oben:= TRUE;
						Abtauen_Heissgas_unten:
							bAbtauen_Heissgas_unten := TRUE;
				END_CASE
				
		END_IF	
	END_IF

END_PROGRAM

// ---- POUs/Funktionen/FB_Schuetzstellung.TcPOU
FUNCTION_BLOCK FB_Schuetzstellung
VAR_INPUT
myStatus: Status_Schuetzstellung;
END_VAR
VAR_OUTPUT
END_VAR
VAR
END_VAR

CASE  myStatus OF

KuehlenOben:
	(*Schütze werden geschaltet*)
		Schuetz_1K3 := TRUE;
		Schuetz_1K4 := FALSE;
		Schuetz_1K5 := TRUE;

	(*Falls Komponente ON ist wird sie auf TRUE gesetzt*)	
		VD_Ventilator_ON			:= TRUE; 
		VD_defrost_Ventilator_ON	:= FALSE;
		ElektrischeHeizung_ON		:= FALSE; 
		KP_ON						:= TRUE;  
		
	(*Expansionsventil wird aktiviert und auf 100% gestellt. Komunikation erfolgt über Modbus_EL*)
	IF  EV.SollKuhlleistung<> 100 THEN 
		EV.SetKuhlleistung := TRUE;
		EV.SollKuhlleistung:= 100;
	END_IF
	
	(*Expansionsventil für die Abtauung wird auf 100% zurückgestellt. Kann verändert werden, um Kälteleistung bzw. Abtaleistung zu variieren*)	
	IF EV_rev.SollKuhlleistung <> 100 THEN 
		EV_rev.SetKuhlleistung := TRUE;
		EV_rev.SollKuhlleistung:= 100;
	END_IF
	
PumpDown: (*Pump-Down wird durchgeführt bis der Druck vor dem KP kleiner als 1,4 Bar ist*)	
	
	(*Schütze werden geschaltet*)
		Schuetz_1K3 := TRUE;
		Schuetz_1K4 := FALSE;
		Schuetz_1K5 := TRUE;
		
	(*Falls Komponente ON ist wird sie auf TRUE gesetzt*)	
		VD_Ventilator_ON			:= FALSE;  //TRUE;
		VD_defrost_Ventilator_ON	:= FALSE;
		ElektrischeHeizung_ON		:= FALSE;
		KP_ON						:= TRUE;  
		
	(*Expansionsventil wird auf 0% gestellt. Komunikation erfolgt über Modbus_EL*)
		EV.SetKuhlleistung := TRUE;
		EV.SollKuhlleistung:= 0;
		
	(*Kompressor PID-Regler wird eingestellt*)
		PID_KP.w := Soll_PumpDownDruck;				//Kompressor wird bei 1.5 Bar ausgeschaltet
		IF  PT_KP_in.rDruck<= Soll_PumpDownDruck THEN 		 
			PID_KP.Aktiv:= FALSE;			 		//Kompressor wird ausgeschaltet
			KP_ON		:= FALSE; 
			
			bPumpDown	:= 	FALSE;					//TRUE-> wird ausgeführt. FALSE-> Beendet/Abgebrochen
			bPumpDownAbgeschlossen:= TRUE; 
		END_IF
		
PumpDown_rev:	(*Schütze, EV_rev werden für PumpDown_rev Modus geschaltet*)

	(*Schütze werden geschaltet*)
		Schuetz_1K3 := FALSE;
		Schuetz_1K4 := TRUE;
		Schuetz_1K5 := FALSE;
		
	(*Falls Komponente ON ist wird sie auf TRUE gesetzt*)	
		VD_Ventilator_ON			:= FALSE;  
		VD_defrost_Ventilator_ON	:= FALSE; //TRUE;
		ElektrischeHeizung_ON		:= FALSE; 
		KP_ON						:= TRUE; 
		
	(*Expansionsventil wird auf 0% gestellt. Komunikation erfolgt über Modbus_EL*)
		EV_rev.SetKuhlleistung := TRUE;
		EV_rev.SollKuhlleistung:= 0;
		
	(*Kompressor PID-Regler wird eingestellt*)
		PID_KP.w := Soll_PumpDownDruck;						//Kompressor wird bei 1.5 Bar ausgeschaltet
		IF PT_KP_in.rDruck<= Soll_PumpDownDruck THEN 
			PID_KP.Aktiv:= FALSE;							//Kompressor wird ausgeschaltet
			KP_ON := FALSE;
			
			bPumpDown_rev := FALSE;							//TRUE-> wird ausgeführt. FALSE-> Beendet/Abgebrochen
			bPumpDown_revAbgeschlossen:= TRUE;
		END_IF
		
AbtauenOben:
	(*Schütze werden geschaltet*)
		Schuetz_1K3 := FALSE;
		Schuetz_1K4 := TRUE;
		Schuetz_1K5 := FALSE;
		
	(*Falls Komponente ON ist wird sie auf TRUE gesetzt*)	
		VD_Ventilator_ON			:= FALSE;  
		VD_defrost_Ventilator_ON	:= TRUE;
		ElektrischeHeizung_ON		:= FALSE; 
		KP_ON						:= TRUE; 
	
AbtauenUnten:
	(*Schütze werden geschaltet*)
		Schuetz_1K3 := FALSE;
		Schuetz_1K4 := FALSE;
		Schuetz_1K5 := FALSE;

	(*Komponente werden de- und aktiviert*)	
		VD_Ventilator_ON			:= FALSE;  
		VD_defrost_Ventilator_ON	:= TRUE;
		ElektrischeHeizung_ON		:= FALSE;
		KP_ON						:= TRUE; 
		
AbtauenElektrisch: 
	(*Schütze werden geschaltet*)
		Schuetz_1K3 := TRUE;
		Schuetz_1K4 := FALSE;
		Schuetz_1K5 := TRUE;

	(*Falls Komponente ON ist wird sie auf TRUE gesetzt*)	
		VD_Ventilator_ON			:= FALSE;  
		VD_defrost_Ventilator_ON	:= FALSE;
		ElektrischeHeizung_ON		:= TRUE; 
		KP_ON						:= FALSE;
		
	(*Expansionsventil wird aktiviert und auf 0% gestellt. Komunikation erfolgt über Modbus_EL*)
		EV.SetKuhlleistung := 	TRUE;
		EV.SollKuhlleistung:= 	0;
	

END_CASE

END_FUNCTION_BLOCK

// ---- POUs/Regelung.TcPOU
PROGRAM Regelung
VAR
	fb_pid_KP : 					CTRL_PID;
	fb_pid_VF : 					CTRL_PID;
	fb_pid_VD_defrost :				CTRL_PID;
	bVF_defrost_TolleranzErreicht: 	BOOL;
	Verzogerungsglied				: FT_PT1;
	Ist_VF_Unterkuhlung_PT1 :		REAL;
END_VAR

(*Soll_zeit für den Automatik-Zyklus Modus wird von Decimal in eine TIME-Variable umgerechnet*)
	IF AutomatikZyklusEin THEN 
	Vereisungszeit := REAL_TO_TIME(DINT_TO_REAL(1000*60)*rVereisungszeit);
	END_IF

(*Stellgrößen werden zugewiesen*)
PID_KP.x:= PT_KP_in.rDruck;				 //PT_KP_in.rDruck; !KP_in Druck funktioniert erst ab < 3 Bar!
PID_VF_Ventilator.x:= PT_VF_out.rDruck;


(*Regler für die Drehzahl des Kompressors*)
IF PID_KP.Aktiv THEN	
fb_pid_KP( 
	ACT:= PID_KP.x, 				//PT.rDruck 
	SET:= PID_KP.w, 				//3.5 [bar]
	SUP:= PID_KP.Einschalttoleranz, 
	OFS:= PID_KP.Offset, 
	M_I:= PID_KP.ManuellerWert, 
	MAN:= PID_KP.ManuellerModus, 
	RST:= bNeuInitialisieren,//PID_KP.Restart, 
	KP:= PID_KP.Kp, 
	TN:= PID_KP.Kp/ PID_KP.I, //2000, 
	TV:= PID_KP.D/ PID_KP.Kp, 
	LL:= Soll_KP.REAL_PARA_minWert,	//PID_KP.LimitUnten, 
	LH:= Soll_KP.REAL_PARA_maxWert,	//PID_KP.LimitOben, 
	Y=> PID_KP.y, 					//4..20mA Kompressor_drehzahl
	DIFF=> PID_KP.e, 
	LIM=> PID_KP.LimitErreicht);
ELSE 
	PID_KP.y := 0; // Regler ist ausgeschalten und sendet 0 mA
END_IF
	Soll_KP.REAL_VAR	 := 		PID_KP.y;	
	
	IF PID_KP.e / PID_KP.w < 0.05 AND -0.05 < PID_KP.e / PID_KP.w THEN 
		bKP_TolleranzErreicht := TRUE;
		ELSE
		bKP_TolleranzErreicht := FALSE;	
	END_IF

	
(*Regler für den Ventilator vom Verflüssiger*)	
Ist_VF_Unterkuhlung := VF.T_v - Temp_VF_out.REAL_VAR;
Verzogerungsglied(In:=Ist_VF_Unterkuhlung, T:=T#10S, K:=1, out=>Ist_VF_Unterkuhlung_PT1);

IF PID_VF_Ventilator.Aktiv THEN	
fb_pid_VF( 
	ACT:= Ist_VF_Unterkuhlung_PT1, 
	SET:= PID_VF_Ventilator.w, // dem Druck entsprechende Verdampfungstemperatur "T_v" minus X Kelvin, garantiert flüssiges Kältemittel im VF-Ausgang
	SUP:= PID_VF_Ventilator.Einschalttoleranz, 
	OFS:= PID_VF_Ventilator.Offset, 
	M_I:= PID_VF_Ventilator.ManuellerWert, 
	MAN:= PID_VF_Ventilator.ManuellerModus, 
	RST:= bNeuInitialisieren,//PID_VF_Ventilator.Restart, 
	KP:= PID_VF_Ventilator.Kp, 
	TN:= PID_VF_Ventilator.Kp/ PID_VF_Ventilator.I, 
	TV:= PID_VF_Ventilator.D/ PID_VF_Ventilator.Kp, 
	LL:= Soll_VF_Ventilator.REAL_PARA_minWert,//PID_VF_Ventilator.LimitUnten, 
	LH:= Soll_VF_Ventilator.REAL_PARA_maxWert,//PID_VF_Ventilator.LimitOben, 
	Y=> PID_VF_Ventilator.y, 
	DIFF=> PID_VF_Ventilator.e, 
	LIM=> PID_VF_Ventilator.LimitErreicht);
ELSE 
	PID_VF_Ventilator.y := 0; // Rergler ist ausgeschaltenen und sendet 0 mA.
END_IF
	Soll_VF_Ventilator.REAL_VAR:= PID_VF_Ventilator.y ;
	
	IF  PID_VF_Ventilator.e / PID_VF_Ventilator.w < 0.05 AND -0.05 < PID_VF_Ventilator.e / PID_VF_Ventilator.w THEN 
		bVF_TolleranzErreicht := TRUE;
		ELSE
		bVF_TolleranzErreicht := FALSE;		
	END_IF

(*!!! Noch nicht impementiert. Verdampfer_defrost wird über Schütz 1K3 direkt mit konstanten 230V versorgt!!

(*Regler für den Ventilator vom Verdampfer außerhalb der Klimakammer in der Abtauphase*)
IF PID_VD_defrost_Ventilator.Aktiv THEN	
fb_pid_VD_defrost( 
	ACT:= PID_VD_defrost_Ventilator.x, 
	SET:= PID_VD_defrost_Ventilator.w, 
	SUP:= PID_VD_defrost_Ventilator.Einschalttoleranz, 
	OFS:= PID_VD_defrost_Ventilator.Offset, 
	M_I:= PID_VD_defrost_Ventilator.ManuellerWert, 
	MAN:= PID_VD_defrost_Ventilator.ManuellerModus, 
	RST:= PID_VD_defrost_Ventilator.Restart, 
	KP:= PID_VD_defrost_Ventilator.Kp, 
	TN:= PID_VD_defrost_Ventilator.Kp/ PID_VD_defrost_Ventilator.I, 
	TV:= PID_VD_defrost_Ventilator.D/ PID_VD_defrost_Ventilator.Kp, 
	LL:= Soll_VD_defrost_Ventilator.REAL_PARA_minWert,//PID_VD_defrost_Ventilator.LimitUnten, 
	LH:= Soll_VD_defrost_Ventilator.REAL_PARA_maxWert,//PID_VD_defrost_Ventilator.LimitOben, 
	Y=> PID_VD_defrost_Ventilator.y, 
	DIFF=> PID_VD_defrost_Ventilator.e, 
	LIM=> PID_VD_defrost_Ventilator.LimitErreicht);
ELSE 
	PID_VD_defrost_Ventilator.y := 0; // Rergler ist ausgeschaltenen und sendet 0 mA ODER 0 V.
END_IF
	Soll_VD_defrost_Ventilator.REAL_VAR:= PID_VD_defrost_Ventilator.y;	
	
	IF PID_VD_defrost_Ventilator.e / PID_VD_defrost_Ventilator.w < 0.05 THEN 
		bVF_defrost_TolleranzErreicht := TRUE;
		ELSE
		bVF_defrost_TolleranzErreicht := FALSE;		
	END_IF
*)

END_PROGRAM

// ---- POUs/Abtauung.TcPOU
PROGRAM Abtauung
VAR
	AbtauFehler : BOOL;
	Timer :TOF;
	Timer_HeizungAbtauwanne: TON;
	
	StartAbtauwanneHeizung : TIME := T#5M; 
	state: INT:= 1;

END_VAR

(*Ablaufstruktur bei einer elektrischen Abtauung des Verdampfers*)
	
	TimerAbtaudauer(IN:=TRUE, PT:= T#1H);
	
	IF bAbtauenAbbrechen = TRUE THEN 
		Mitteilung 				:= 'Abtauvorgang wurde abgebrochen!';
		bLeerlauf				:=TRUE;
		bKuehlen 				:=FALSE;
		bAbtauen				:=FALSE;
		bAbtauen_elektrisch		:=FALSE;
			ElektrischeHeizung_ON := FALSE;
		bAbtauen_Heissgas_oben	:=FALSE;
		bAbtauen_Heissgas_unten	:=FALSE;
		bPumpDownAbgeschlossen := FALSE;
		TimerAbtaudauer			(IN:= FALSE);
		state					:= 0;
	(*nächster Status*)
		SM.Status := Leerlauf;
	
		ELSE 
		bLeerlauf :=FALSE; 
	END_IF

CASE state OF
	
		
0: 
	bAbtauenAbgeschlossen := FALSE;
	
	(*Regler werden ausgeschaltet*)
	
		PID_KP.Aktiv:= 					FALSE;
		PID_VF_Ventilator.Aktiv :=		FALSE;
		VD_Ventilator_ON:= 				FALSE;
		VD_defrost_Ventilator_ON := 	FALSE;
		KP_ON:= 						FALSE;
	(*Nächster State wird je nach Abtau-Modus ausgewählt*)	
		IF bAbtauen_elektrisch THEN
		state:= 1;
		END_IF	
		
		IF bAbtauen_Heissgas_oben THEN
		state:= 5;
		END_IF	
		
		IF bAbtauen_Heissgas_unten THEN
		state:= 5;
		END_IF	
		
		IF NOT bAbtauen_elektrisch AND NOT bAbtauen_Heissgas_oben AND NOT bAbtauen_Heissgas_unten THEN
		AbtauFehler := TRUE;
		state:= 0;
		ELSE 
		AbtauFehler := FALSE;
		END_IF
			
1:	
	(*Elektrische Heizung wird eingeschaltet*)
		ElektrischeHeizung_ON := TRUE;								// Schütz wird geschaletet und Heizung kann nun geregelt werden
		Timer_HeizungAbtauwanne(In:= TRUE, PT:= StartAbtauwanneHeizung);
		
		(*Ausgewählte Heizleistung für Bodenheizung und Heizracks*)
		//Regler aktivieren
			Soll_ElektHeizrack1.REAL_VAR := 	 Heizstufe;
			Soll_ElektHeizrack2.REAL_VAR := 	 Heizstufe;
		IF Timer_HeizungAbtauwanne.Q THEN
			Soll_ElektHeizrack_Boden.REAL_VAR := Heizstufe;
		END_IF

		(*Berechnet die tatsächliche Leistung*)
			P_el_Boden:= Heizstufe/10	*P_el_Boden_max;
			P_el_Rack1:= Heizstufe/10	*P_el_Rack_max;
			P_el_Rack2:= Heizstufe/10	*P_el_Rack_max;	

		(*Gesamte Heizleistung wird berechnet*)
			P_el_Heizung_ges:= P_el_Boden + P_el_Rack1 + P_el_Rack2;

	
	(*Überprüfung ob Oberflächentemperatur auf dem Verdampfer größer als 10°C ist*)
	(*Elektrische Heizung wird ausgeschaltet*)

		IF 	Temp_VD_Surface_gemittelt > 10 THEN
			ElektrischeHeizung_ON := FALSE;
			Timer_HeizungAbtauwanne(In:= FALSE);  		//Reset Timer
			Soll_ElektHeizrack1.REAL_VAR := 	0;		// Ausschalten der Heizung
			Soll_ElektHeizrack2.REAL_VAR := 	0;		// Ausschalten der Heizung
			Soll_ElektHeizrack_Boden.REAL_VAR :=0;		// Ausschalten der Heizung
			
			state:= 8;	
		END_IF


5:
	(*state wird je nach Methode gewählt*)	
		IF bAbtauen_Heissgas_oben THEN 
			state:= 6;
		END_IF
		
		IF bAbtauen_Heissgas_unten THEN 
			state:=7; 
		END_IF
		
6: 	
	(*Schalte auf Abtauen von Oben*)
		fb_Schuetzstellung(myStatus:= AbtauenOben);
		
		state:= 8;
	
7:	
	(*Schalte auf Abtauen von Unten*)
		fb_Schuetzstellung(myStatus:= AbtauenUnten);
						
		state:=8;

8: 	
	(*Kompressor und Ventilator vom VD_defrost werden eingeschaltet*)		
		KP_ON:= 					TRUE;
		PID_KP.Aktiv :=				TRUE;
		VD_defrost_Ventilator_ON := TRUE;
		
		IF Temp_VD_Surface_gemittelt > 10 THEN			
			KP_ON:= 					FALSE;
			PID_KP.Aktiv := 			FALSE;
			VD_defrost_Ventilator_ON := FALSE;
			state:= 9;
			Timer(IN:=FALSE);
		END_IF
9: 
	(*Starte Timer. Timer läuft 10 Minuten*)
		Timer(IN:= TRUE, PT:= T#10M);
	
		IF Timer.Q THEN
			state:= 10;
			Timer(IN:= FALSE);
		END_IF
	
10: 	
	(*Schalte Schütze auf Kühlen*)
		fb_Schuetzstellung(myStatus:= KuehlenOben);
	
	(*Kompressor wird eingeschaltet*)
		KP_ON		:= TRUE;
		PID_KP.Aktiv:= TRUE;
		
	(*Überprüfung ob Oberflächentemperatur auf dem Verdampfer kleiner als 0°C ist*)	
		IF Temp_VD_Surface_gemittelt< 0 THEN
			VD_Ventilator_ON:= TRUE;
			state:=11;
		END_IF
		
11: 	
	(*Anlage wird reverse abgepumpt, falls sie zuvor per Heißgas(oben oder unten) abgetaut wurde*)	
		IF bAbtauen_Heissgas_oben = TRUE OR bAbtauen_Heissgas_unten = TRUE THEN 
		 bPumpDown_rev := TRUE;
		END_IF

	(*Abtau-Vorgang ist abgeschlossen. State-Maschine: Abtauen->FALSE. Kuehlen-> TRUE. *)	
		Mitteilung:= 				'Abtau-Vorgang wurde erfolgreich abgeschlossen';
		bAbtauenAbgeschlossen := 	TRUE;
		bAbtauen			:= 		FALSE;
		bAbtauen_elektrisch:= 		FALSE;
		bAbtauen_Heissgas_oben:= 	FALSE;
		bAbtauen_Heissgas_unten:= 	FALSE;
		bPumpDownAbgeschlossen := 	FALSE;
	(*Kühl-Modus wird aktiviert und gegebenfalls ein PUMPDOWN_rev durchgeführt*)
		IF AutomatikZyklusEin THEN 
				bKuehlen:= TRUE;
				CASE  AutomatikAbtauModus OF 
						NichtAusgewahlt: 
							Mitteilung := 'Kein Automatik-Abtaumodus ausgewählt!';
						Abtauen_elektrisch:
							bPumpDown_rev := FALSE;
						Abtauen_Heissgas_oben:
							bPumpDown_rev:= TRUE;
						Abtauen_Heissgas_unten:
							bPumpDown_rev := TRUE;
				END_CASE
		END_IF
		
	(*Gestoppte Zeit für den Abtauzyklus wird auf Null gesetzt*)
		TimerAbtaudauer(IN:= FALSE);
	
	(*Reset von State auf Null*)
		state:= 0;
	
		
END_CASE

END_PROGRAM

// ---- POUs/Anlagenschutz/Kompressorschutz.TcPOU
PROGRAM Kompressorschutz
VAR
	BerechneT_Taulinie: FB_GetEnthalpie;
	Temp_Taulinie :REAL;
END_VAR

(*Kompressor läuft langsam an, um möglichen Tropfenschlag zu verhindern. Überhitzungstemperatur im 
  Expansionsventil wird überprüft*)


(*Unterdurckschutz. Kompressor wird ausgeschaltet*) 
IF PT_KP_in.rDruck < 1.0 THEN
	 Soll_KP.REAL_VAR := 0;
	 KP_ON := FALSE;			
	 SM.Mitteilung := 'Unterdruckschutz wurde aktiviert';
END_IF

(*Überdruckschutz. Kompressor wird ausgeschaltet*) 
IF PT_KP_out.rDruck > 15 THEN
	 Soll_KP.REAL_VAR := 0;
	 KP_ON := FALSE;
	 SM.Mitteilung := 'Überdruckschutz wurde aktiviert';
END_IF


(*Beim PUMPDOWN wird das Kältemittel vor dem Kompressor sehr kalt. Kompressor wird ausgeschaltet, wenn
 die Temperatur vor dem Kompressor nur noch 2 K wärmer als die Taulinie ist*)
 BerechneT_Taulinie(In_Druck:= KP.p_in, In_Temperatur := KP.T_in, T_v=> Temp_Taulinie) ;
 
(*
 IF KP.T_in < Temp_Taulinie-2 AND (bPumpDown OR bPumpDown_rev)  THEN 
	 KP_ON 		  := FALSE;
	 Soll_KP.REAL_VAR := 0;
	  SM.Mitteilung := 'Die Temperatur vor Kompressor ist zu kalt. Kompressor enthält keine Freigabe.';
 END_IF
 
*)

END_PROGRAM

// ---- POUs/Anlagenschutz/Sonstiges.TcPOU
PROGRAM Sonstiges
VAR
END_VAR

(*Eingabewerte von Soll_Heizungswerte werden begrenzt, damit sie zwischen 0..10 V liegen*)
	Soll_ElektHeizrack1.REAL_VAR := 	  LIMIT(Soll_ElektHeizrack1.REAL_PARA_minWert ,Heizstufe,Soll_ElektHeizrack1.REAL_PARA_maxWert);
	Soll_ElektHeizrack2.REAL_VAR := 	  LIMIT(Soll_ElektHeizrack2.REAL_PARA_minWert,Heizstufe,Soll_ElektHeizrack2.REAL_PARA_maxWert);
	Soll_ElektHeizrack_Boden.REAL_VAR :=  LIMIT(Soll_ElektHeizrack_Boden.REAL_PARA_minWert,Heizstufe,Soll_ElektHeizrack_Boden.REAL_PARA_maxWert);
	
(*Überhitzungsschutz für Verdampfer.*)
	IF Temp_VD_Surface_gemittelt > 80 THEN 
		bAbtauen_elektrisch := FALSE;
		bAbtauen_Heissgas_oben:= FALSE;
		bAbtauen_Heissgas_unten:=FALSE;
		Mitteilung:= 'Überhitzungsschutz vom Verdampfer ist aktiviert worden';
		WarnungAnlagenschutz	 := TRUE;
	END_IF
	
(*Waagenschutz. Waagen sind nur bis 10 kg belastbar. Weitere Belastungen könnten zu Beschädigungen der Waagen führen.
  In diesem Fall wird abgetaut und der Verdampfer vom Eis befreit. Die Waagen werden entlastet. *)
  
  IF Waage_roh[1]> 10000 OR Waage_roh[2] >10000 OR Waage_roh[3] >10000 OR Waage_roh[4] >10000 OR Waage_roh[5] >10000 OR Waage_roh[6] >10000 THEN 
	  WarnungAnlagenschutz	 := TRUE;
	  Mitteilung := 'Waagenschutz ist aktiviert worden'; 
	  
	  bAbtauen := TRUE;
	  bAbtauen_elektrisch:= TRUE;
	  
	  //Vereisungsprozess wird abgebrochen
	  bKuehlenAbbrechen := TRUE;
  END_IF
  
  
(*Elektrische Heizung Schutz. Falls ElektrischeHeizung_ON nicht TRUE werden auch alle AO-Ausgangssignale 
  der Heizungsregelung auf 0 V gestellt*)
  
  		IF ElektrischeHeizung_ON = FALSE THEN 
			Soll_ElektHeizrack1.REAL_VAR		:= 0;
			Soll_ElektHeizrack2.REAL_VAR		:= 0;
			Soll_ElektHeizrack_Boden.REAL_VAR 	:= 0;
		END_IF

END_PROGRAM

// ---- POUs/SchreibeSollwerte.TcPOU
PROGRAM SchreibeSollwerte
VAR
END_VAR

CASE SM.Status OF
	
	Lesen:
	
	
	Schreiben:
	
	//Stellsignal Veflüssiger Ventilator
		Soll_VF_Ventilator.INT_VAR_Output:=	FB_Nativ_zu_SPS_lin(output:=Soll_VF_Ventilator);

	//Stellsignal Kompressor
		Soll_KP.INT_VAR_Output:= 			FB_Nativ_zu_SPS_lin(output:=Soll_KP);
	
	//Stellsignal elektrische Heizung

		Soll_ElektHeizrack1.INT_VAR_Output		:= FB_Nativ_zu_SPS_lin(output:= Soll_ElektHeizrack1);
		Soll_ElektHeizrack2.INT_VAR_Output		:= FB_Nativ_zu_SPS_lin(output:= Soll_ElektHeizrack2);
		Soll_ElektHeizrack_Boden.INT_VAR_Output := FB_Nativ_zu_SPS_lin(output:= Soll_ElektHeizrack_Boden);
		
	// DIgitale Ausgänge werden zugeordnet
		DO_VD_Ventilator_ON 		:= VD_Ventilator_ON;
		DO_VD_defrost_Ventilator_ON := VD_defrost_Ventilator_ON;
		DO_ElektrischeHeizung_ON 	:= ElektrischeHeizung_ON ;
		DO_KP_ON 					:= KP_ON;	
		DO_Schuetz_1K3 				:= Schuetz_1K3 	;
		DO_Schuetz_1K4				:= Schuetz_1K4	;
		DO_Schuetz_1K5				:= Schuetz_1K5;
END_CASE

END_PROGRAM

// ---- POUs/Funktionen/FB_Nativ_zu_SPS_lin.TcPOU
FUNCTION FB_Nativ_zu_SPS_lin : int
VAR_INPUT
	output:output_var;
END_VAR
VAR
END_VAR

FB_Nativ_zu_SPS_lin:=  real_to_int((output.REAL_VAR-output.REAL_PARA_C)/output.REAL_PARA_M);

END_FUNCTION

// ---- POUs/Waagen/Hintergrund.TcPOU
PROGRAM Hintergrund
VAR   
 (* background communication with the EL6002 terminal *)
 	fbEL6002Ctrl: 		ARRAY[1..6] OF SerialLineControl;
 	bEL6002CtrlError: 	ARRAY[1..6] OF BOOL;
	eEL6002CtrlErrorID: ARRAY[1..6] OF ComError_t;
	counter: INT;
END_VAR


IF counter >= 6 THEN 
	counter:= 1;
END_IF

//--Jede Waage wird abgefragt. Der counter läuft einmal durch und fragt jeweils den neuesten Datenstring ab.

FOR counter:= 1 TO 6 DO
fbEL6002Ctrl[counter](   
	Mode:= 		SERIALLINEMODE_EL6_22B, 
   pComIn:= 	ADR(Waage[counter].EL6002_in), 
   pComOut:= 	ADR(Waage[counter].EL6002_out), 
   SizeComIn:=	SIZEOF(Waage[counter].EL6002_in), 
   Error=> 		bEL6002CtrlError[counter], 
   ErrorID=> 	eEL6002CtrlErrorID[counter], 
   TxBuffer:= 	TxBuffer[counter], 
   RxBuffer:= 	RxBuffer[counter] );
END_FOR

END_PROGRAM

// ---- POUs/Datenbank/DB_Lesen_Stoffwerte_Wasser.TcPOU
PROGRAM DB_Lesen_Stoffwerte_Wasser
VAR

	  
   //FB_DB_Schliesse_PID:FB_DBConnectionClose;

	DB_Stoffwerte_Wasser: ARRAY[0..100] OF ST_DB_STOFFWERTE;	

	FB_DB_Lese_Dampftafel: FB_DBRecordArraySelect;
	sSelectString: STRING(800):= 'SELECT 	`id`,	`temp`,	`dichte` , `cp` FROM	`stoffwerte_wasser`';
	nRecIndex: UDINT;
	bStartStopSelect: BOOL;
	bBusySelect: BOOL;
	bErrorSelect: BOOL;
	stSQLStateSelect: TC2_DATABASE.ST_DBSQLError;
	nRecordCount: UDINT;
	Busy_Lesen:BOOL;
	start_Lesen:BOOL:=TRUE;
	start_Schliessen:BOOL:=FALSE;
	Counter: UDINT:=0;
	
	pCmdAddr: UDINT;
	
END_VAR

IF 	SM.Leerlauf THEN
	
start_Lesen:=TRUE;
SM.Leerlauf:=FALSE;
	
END_IF

//=========================================================================================	
//Dampftafel auslesen		
	FB_DB_Lese_Dampftafel(
				sNetID:=, 
				hDBID:= 7, 
				pCmdAddr:= ADR(sSelectString), 
				cbCmdSize:= SIZEOF(sSelectString), 
				nStartIndex:= nRecIndex, 
				nRecordCount:=nRecordCount-1, 
				pDestAddr:= ADR(DB_Stoffwerte_Wasser), 
				cbRecordArraySize:= SIZEOF(DB_Stoffwerte_Wasser), 
				bExecute:= start_Lesen, 
				tTimeout:= T#5S, 
				bBusy=> Busy_Lesen, 
				bError=> SM.bDBFehler, 
				nErrID=> , 
				sSQLState=> stSQLStateSelect, 
				nRecords=> nRecordCount); 
				

				
	IF Busy_Lesen=FALSE THEN
			start_Lesen:=FALSE;
		start_Schliessen:=TRUE;
	END_IF
	
	(*FB_DB_Schliesse_PID(
				sNetID:= , 
				hDBID:=3, 
				bExecute:= start_Schliessen_PID, 
				tTimeout:= T#1S, 
				bBusy=> , 
				bError=> SM.Fehler, 
				nErrID=> );
	
	*)
	
	IF nRecordCount>0 THEN
		
		FOR counter:=0 TO nRecordCount-1 BY 1 DO
	   
	HYD.Stoffwerte_Wasser[counter].Temperatur :=STRING_TO_REAL(DB_Stoffwerte_Wasser[counter].temp);
	HYD.Stoffwerte_Wasser[counter].Dichte :=STRING_TO_REAL(DB_Stoffwerte_Wasser[counter].dichte);
	HYD.Stoffwerte_Wasser[counter].cp :=STRING_TO_REAL(DB_Stoffwerte_Wasser[counter].cp);		
		
		END_FOR
	END_IF
	
	
	IF Busy_Lesen=FALSE AND nRecordCount>0 THEN
		SM.Leerlauf:=TRUE;
		ELSE  sm.Leerlauf:=FALSE;
	END_IF

END_PROGRAM

// ---- POUs/Funktionen/CTLR_PID_Negativ.TcPOU
FUNCTION_BLOCK CTLR_PID_Negativ
VAR_INPUT
	ACT, SET, SUP, OFS, M_I : REAL;
	MAN : BOOL;
	RST : BOOL;
	KP : REAL := 1.0;
	TN : REAL := 1.0;
	TV : REAL := 1.0;
	LL : REAL := -1000.0;
	LH : REAL := 1000.0;
END_VAR
VAR_OUTPUT
	Y : REAL;
	DIFF : REAL;
	LIM : BOOL;
END_VAR
VAR
	pid : FT_PIDWL;
	co : CTRL_OUT;
END_VAR



(*
version 2.0	30. jun. 2008
programmer 	hugo
tested by	oscat

FT_PI is a PI controller with manual functionality.
The PID controller works according to the fomula Y = e *(KP+ KI * INTEG(e) ) + offset, while e = set_point - actual.
a rst will reset all internal data, while a switch to manual will cause the controller to follow the function Y = manual_in + offset.
limit_h and Limit_l set the possible output range of Y.
the output flags lim will signal that the output limits are active.

*)

DIFF := CTRL_IN(SET, ACT, SUP);
pid(in := -DIFF, kp := KP, tn := TN, tv := TV, lim_l := LL, lim_h := LH, rst := RST);
co(ci := pid.Y, OFFSET := OFS, man_in := M_I, lim_l := LL, lim_h := LH, MANUAL := MAN);
Y := co.Y;
LIM := co.LIM;



(* revision history

hm 1.12.2006	 	rev 1.1
	changed algorithm to trapezregel for higher accuracy.

hm 3.1.2007		rev 1.2
	added integ_band to select when the integrator is active.

hm	3.3.2007		rev 1.3
	added default values to inputs KP, TN, TV, LIMIT_L und LIMIT_H.

hm 31.oct 2007	rev 1.4
	total rewrite of the module to avoid failures when one of the limits is 0

hm	3.11.2007	rev 1.5
	added noise input to filter noise
	added output diff
	set limit output false when output is within limits
	overfolw was not set correctly

hm	5. jan 2008	rev 1.6
	improved code for better performance
	
DIFF:= -DIFF; 
*)

END_FUNCTION_BLOCK

// ---- POUs/Funktionen/FB_PT1.TcPOU
FUNCTION FB_PT1 : Input_Var
VAR_INPUT
	mInput_Var:INPUT_VAR;
	
	
END_VAR
VAR
pt1:FT_PT1;
END_VAR

pt1(in:=mInput_Var.REAL_VAR,T:=mInput_Var.REAL_PARA_PT1_T,K:=mInput_Var.REAL_PARA_PT1_K,out=>mInput_Var.REAL_VAR_PT1);
FB_PT1:=mInput_Var;

END_FUNCTION

// ---- POUs/Funktionen/FB_SPS_zu_Nativ_INPUT_VAR.TcPOU
FUNCTION FB_SPS_zu_Nativ_INPUT_VAR : INPUT_VAR
VAR_INPUT
	INPUT: INPUT_VAR;
	
END_VAR
VAR
END_VAR

//Lineare Umrechnung der Eingangsgröße vom Typ INT in den nativen Wert vom Typ REAL
INPUT.REAL_VAR := INPUT.REAL_PARA_M * INPUT.INT_VAR_Input + INPUT.REAL_PARA_C;

//Übergabe an den Rückgabewert
FB_SPS_zu_Nativ_INPUT_VAR:=INPUT;

END_FUNCTION

// ---- POUs/Funktionen/POU.TcPOU
FUNCTION_BLOCK POU
VAR_INPUT
END_VAR
VAR_OUTPUT
END_VAR
VAR
END_VAR

END_FUNCTION_BLOCK

// ---- POUs/Funktionen/FB_PID.TcPOU
FUNCTION_BLOCK FB_PID //EXTENDS CTRL_PID
VAR_INPUT
	PID_in : PID;
END_VAR
VAR_OUTPUT
	PID_out: PID;
END_VAR
	
VAR
	FB_PID: CTRL_PID;
END_VAR

IF PID_in.Aktiv THEN

	FB_PID( 
	ACT:= PID_in.x, 
	SET:= PID_in.w, 
	SUP:= PID_in.Einschalttolleranz, 
	OFS:= PID_in.Offset, 
	M_I:= PID_in.ManuellerWert, 
	MAN:= PID_in.ManuellerModus, 
	RST:= PID_in.Restart, 
	KP:= PID_in.Kp, 
	TN:= PID_in.Kp/ PID_in.I, 
	TV:= PID_in.D/ PID_in.Kp, 
	LL:= PID_in.Limit_unten, 
	LH:= PID_in.Limit_oben, 
	Y=> PID_in.y, 
	DIFF=> PID_in.e, 
	LIM=> PID_in.LimitErreicht);
ELSE 
	// Rergler ist ausgeschaltenen und sendet 0 mA ODER 0 V.
	PID_in.y := 0; 
END_IF

PID_out:= PID_in;

END_FUNCTION_BLOCK

// ---- POUs/Funktionen/WORD_TO_BINSTRING.TcPOU
FUNCTION WORD_TO_BINSTRING : STRING(16)
VAR_INPUT
	myWORD:DWORD;		//WORD aus der Klemme/Modbusarray
END_VAR
VAR
		b1: BYTE;
		b0: BYTE;

		s1: STRING(8);
		s0: STRING(8);
END_VAR

(*da Twincat mit LIL-Endian arbeitet und die Kellersensoren mit BIG-Endian,
 müssen die Bytes paarweise vertauscht werden*)

//Zerteilen des DWORDs in die 4 Bytes

b1:= BYTE_OF_DWORD(myWORD, 0);
b0:= BYTE_OF_DWORD(myWORD, 1);

//Umrechnung der BYTES in Binärestrings mit der Länge 8 bits

s1:= BYTE_TO_BINSTR(b1,8);
s0:= BYTE_TO_BINSTR(b0,8);

//Zusammenfügen der vier Binärstrings zu einem 32 bit String
DWORD_TO_BINSTRING := CONCAT(s1,s0);

END_FUNCTION

// ---- POUs/Modbus/ConfigMassenstromsensor.TcPOU
PROGRAM ConfigMassenstromsensor
VAR
	state : INT := 1;
	
	baudrate_neu:	 	LINT;
	baudrate_alt:	 	LINT;
	baudrate_lilendian: LINT;
	
	ModbusAdresse_alt: 	 BYTE := 12;	//Massenstromsensor hat die default-Adresse 1
	ModbusAddress_neu: 	 BYTE := 12; //Massenstromsensor hat die Adresse 12 im ModbusRTU
	
	Parity_alt: 			ARRAY[0..1]OF BYTE ;
	Parity_neu:				ARRAY[0..1]OF BYTE := [3,0];
	
	RegisterFormat_alt:			ARRAY[0..1]OF BYTE :=[1, 0]; // in Big Endian
	RegisterFormat_neu:			ARRAY[0..1]OF BYTE :=[0, 0]; // in Big Endian
	
	
	

END_VAR

CASE MODBUS.Status_Modbus OF

ConfigMSS:
	
	CASE state OF
		
		1:
		
		MODBUS.myModbus.ReadRegs( 		 
			UnitID:= ModbusAdresse_alt,
 			 Quantity:= 2,
 			 MBAddr:= 50000,						
 			 cbLength:= SIZEOF(baudrate_alt),
 			 pMemoryAddr:= ADR(baudrate_alt),
  			Execute:= TRUE,
  			Timeout:= modbusTimeout,
  			Busy => isModbusBusy,
  			Error => isModbusError,
  			ErrorId => modbusErrorId
  			(* cbRead parameter *));
			
		
		IF NOT isModbusBusy THEN
				MODBUS.myModbus.ReadRegs(Execute:= FALSE);
				IF MODBUS.myModbus.Error THEN
				state := 1;
				ELSE
				state := 1;	
			END_IF
		END_IF
		
		baudrate_lilendian:= BE32_TO_HOST(LINT_TO_DWORD( baudrate_alt));
		
(*
	2:
		MODBUS.myModbus.WriteRegs( 		 
			UnitID:= ModbusAdresse,
 			Quantity:= 2,
 			MBAddr:= 50004,						
 			cbLength:= SIZEOF(baudrate_alt),
 			pMemoryAddr:= ADR(baudrate_alt),
  			Execute:= TRUE,
  			Timeout:= modbusTimeout,
  			Busy => isModbusBusy,
  			Error => isModbusError,
  			ErrorId => modbusErrorId
  			(* cbRead parameter *));
			
		
		IF NOT isModbusBusy THEN
				MODBUS.myModbus.WriteRegs(Execute:= FALSE);
				IF MODBUS.myModbus.Error THEN
				state := 1;
				ELSE
				state := 32;	
			END_IF
		END_IF
*)
		
	END_CASE
	
END_CASE

END_PROGRAM

// ---- POUs/Testprogramme/Druckumrechnung.TcPOU
PROGRAM Druckumrechnung
VAR
	
	fbton1: TON;
	flag: BOOL := TRUE;
	stDruck		:DWORD:= 10000001001010010000001011011110;
	stDruck2: T_MaxString;
	stByte_reg1: STRING;
	stByte_reg2: STRING;
	stReg: T_MaxString;
	stReg1: STRING;
	stReg2: STRING;
	DruckBaby: LREAL;
	Reg: T_FIX16;
	
	stSign		:STRING(255);
	iSign		:INT;
	stExponent	:STRING(255);
	iExponent	:INT;	
	stMantis	:STRING(255);
	iMantis		:INT;
	rMantis		:REAL;// := 2687710;
	fDruck		:LREAL;
	rSign: REAL ;//:= 0;
	rExponent: REAL ;// := 130;
	Test: REAL2;
	rTest: REAL;
	DWSign: DWORD;
	DWExponent: DWORD;
	DWMantis: DWORD;
	Var1: WORD;

	
	
END_VAR

//		fbton1(IN:= NOT fbton1.Q, PT:= T#1S, Q=> , ET=> );

(*
Byte_reg1 := BE32_TO_HOST(in:= modbusData[20]);
Reg:=WORD_TO_FIX16(in:=modbusData[20],n:= 15 );
DruckBaby:=FIX32_TO_LREAL(in:=Reg)*100;
*)

(*
Byte_reg1 := BE16_TO_HOST(in:= modbusData[20]);
Byte_reg2 := BE16_TO_HOST(in:= modbusData[21]);

stByte_reg1 := WORD_TO_BINSTR (in:=Byte_reg1, iPrecision :=16);
stByte_reg2 := WORD_TO_BINSTR (in:=Byte_reg2, iPrecision :=16);

stDruck:= CONCAT(STR1:= stByte_reg1, STR2:= stByte_reg2);

*)

//stDruck:=DWORD_TO_BINSTR(in:= BE32_TO_HOST(in:= modbusData[20]), iPrecision:=32);




stSign:= LEFT(stDruck,1);
iSign:=LEN(stSign);
DWSign:=BIN_TO_DWORD(BIN:= stSign);
rSign:= DWORD_TO_REAL(DWSign);
		
		
stExponent	:=RIGHT(LEFT(stDruck,9),8);
iExponent	:=LEN(stExponent);
DWExponent	:=BIN_TO_DWORD(BIN:=stExponent);
rExponent	:= DWORD_TO_REAL(DWExponent);

stMantis	:= RIGHT(stDruck,23);
iMantis		:= LEN(stMantis);
DWMantis	:= BIN_TO_DWORD(BIN:=stMantis);
rMantis		:= DWORD_TO_REAL (DWMantis);

fDruck := F_POWER(a:= 1, x:= (-1), n:= rSign)*(1+ rMantis/8388608)* F_POWER(a:=1, x:= 2, n:=(rExponent-127));

END_PROGRAM

// ---- POUs/Testprogramme/FB_FileCopy.TcPOU
FUNCTION_BLOCK FB_FileCopy
VAR_INPUT
    sSrcNetId            : T_AmsNetID;
    sSrcPathName         : T_MaxString;
    sDestNetId           : T_AmsNetId;
    sDestPathName        : T_MaxString;
    bExecute             : BOOL;
    tTimeOut             : TIME := DEFAULT_ADS_TIMEOUT;
END_VAR
VAR_OUTPUT
    bBusy                : BOOL;
    bError               : BOOL;
    nErrId               : UDINT;
END_VAR
VAR
    fbFileOpen           : FB_FileOpen;
    fbFileClose          : FB_FileClose;
    fbFileRead           : FB_FileRead;
    fbFileWrite          : FB_FileWrite;
    hSrcFile             : UINT := 0;(* File handle of the source file *)
    hDestFile            : UINT := 0;(* File handle of the destination file *)

    Step                 : DWORD;
    RisingEdge           : R_TRIG;
    buffRead             : ARRAY[1..1000] OF BYTE;(* Buffer *)
    cbReadLength         : UDINT := 0;
END_VAR

RisingEdge(CLK:=bExecute); 
 
CASE Step OF 
     0:     (* Idle state *) 
          IF RisingEdge.Q THEN 
               bBusy := TRUE; 
               bError:= FALSE; 
               nErrId:=0; 
               Step := 1; 
               cbReadLength:=0; 
               hSrcFile:=0; 
               hDestFile:=0; 
          END_IF 
 
     1:     (* Open source file *) 
          fbFileOpen( bExecute := FALSE ); 
          fbFileOpen( sNetId := sSrcNetId, sPathName := sSrcPathName, 
                         nMode := FOPEN_MODEREAD OR FOPEN_MODEBINARY, 
                         ePath := PATH_GENERIC, tTimeout := tTimeOut, bExecute := TRUE ); 
          Step := Step + 1; 
     2: 
          fbFileOpen( bExecute := FALSE ); 
          IF NOT fbFileOpen.bBusy THEN 
               IF fbFileOpen.bError THEN 
                    nErrId := fbFileOpen.nErrId; 
                    bError := TRUE; 
                    Step := 50; 
               ELSE 
                    hSrcFile := fbFileOpen.hFile; 
                    Step := Step + 1; 
               END_IF 
          END_IF 
 
     3:     (* Open destination file *) 
          fbFileOpen( bExecute := FALSE ); 
          fbFileOpen( sNetId := sDestNetId, sPathName := sDestPathName, 
                         nMode := FOPEN_MODEWRITE OR FOPEN_MODEBINARY, 
                         ePath := PATH_GENERIC, tTimeout := tTimeOut, bExecute := TRUE ); 
          Step := Step+1; 
     4: 
          fbFileOpen( bExecute := FALSE ); 
          IF NOT fbFileOpen.bBusy THEN 
               IF fbFileOpen.bError THEN 
                    nErrId := fbFileOpen.nErrId; 
                    bError := TRUE; 
                    Step := 50; 
               ELSE 
                    hDestFile := fbFileOpen.hFile; 
                    Step := Step + 1; 
               END_IF 
          END_IF 
 
     5:     (* Read data from source file *) 
          cbReadLength := 0; 
          fbFileRead( bExecute:= FALSE ); 
          fbFileRead( sNetId:=sSrcNetId, hFile:=hSrcFile, 
                         pReadBuff:= ADR(buffRead), cbReadLen:= SIZEOF(buffRead), 
                         bExecute:=TRUE, tTimeout:=tTimeOut ); 
          Step := Step + 1; 
     6: 
          fbFileRead( bExecute:= FALSE ); 
          IF NOT fbFileRead.bBusy THEN 
               IF fbFileRead.bError THEN 
                    nErrId := fbFileRead.nErrId; 
                    bError := TRUE; 
                    Step := 50; 
               ELSE 
                    cbReadLength := fbFileRead.cbRead; 
                    Step := Step + 1; 
               END_IF 
          END_IF 
 
     7:     (* Write data to destination file *) 
          fbFileWrite( bExecute := FALSE ); 
          fbFileWrite( sNetId:=sDestNetId, hFile:=hDestFile, 
                         pWriteBuff:= ADR(buffRead), cbWriteLen:= cbReadLength, 
                         bExecute:=TRUE, tTimeout:=tTimeOut ); 
          Step := Step + 1; 
     8: 
          fbFileWrite( bExecute := FALSE ); 
          IF NOT fbFileWrite.bBusy THEN 
               IF fbFileWrite.bError THEN 
                    nErrId := fbFileWrite.nErrId; 
                    bError := TRUE; 
                    Step := 50; 
               ELSE 
                    IF fbFileRead.bEOF THEN (* Check if the EOF flag ist set *) 
                         Step := 50;     (* Cleanup: close the destination and source files *) 
                    ELSE 
                         Step := 5; (* Repeat reading/writing *) 
                    END_IF 
               END_IF 
          END_IF 
 
     30:     (* Close the destination file *) 
          fbFileClose( bExecute := FALSE ); 
          fbFileClose( sNetId:=sDestNetId, hFile:=hDestFile, bExecute:=TRUE, tTimeout:=tTimeOut ); 
          Step := Step + 1; 
     31: 
          fbFileClose( bExecute := FALSE ); 
          IF NOT fbFileClose.bBusy THEN 
               IF fbFileClose.bError THEN 
                    nErrId := fbFileClose.nErrId; 
                    bError := TRUE; 
               END_IF 
               Step := 50; 
               hDestFile := 0; 
          END_IF 
 
     40: (* Close source file *) 
          fbFileClose( bExecute := FALSE ); 
          fbFileClose( sNetId:=sSrcNetId, hFile:=hSrcFile, bExecute:=TRUE, tTimeout:=tTimeOut ); 
          Step := Step + 1; 
     41: 
          fbFileClose( bExecute := FALSE ); 
          IF NOT fbFileClose.bBusy THEN 
               IF fbFileClose.bError THEN 
                    nErrId := fbFileClose.nErrId; 
                    bError := TRUE; 
               END_IF 
               Step := 50; 
               hSrcFile := 0; 
          END_IF 
 
     50: (* Error or ready => Cleanup *) 
          IF ( hDestFile <> 0 ) THEN 
               Step := 30; (* Close the destination file*) 
          ELSIF (hSrcFile <> 0 ) THEN 
               Step := 40; (* Close the source file *) 
          ELSE 
               Step := 0;     (* Ready *) 
               bBusy := FALSE; 
          END_IF 
 
END_CASE

END_FUNCTION_BLOCK

// ---- POUs/Testprogramme/FB_SerialCom.TcPOU
FUNCTION_BLOCK FB_SerialCom
VAR_IN_OUT
	TxBuffer: ComBuffer;
END_VAR

VAR
	Timer: TP;
	fbSend : SendString;
	fbReceive: ReceiveString;
	bSendBusy: BOOL := FALSE;
	eSendErrorID: ComError_t;
	sReceivedString: STRING;
	bStringReceived: BOOL;
	bReceiveBusy: BOOL;
	eReceiveErrorID: ComError_t;
	bReceiveTimeout: BOOL;
	nReceiveCounter: INT;
	sLastReceiveString: STRING;
	ClearComBuffer : ClearComBuffer;
END_VAR

Timer(IN:=TRUE,PT:= T#10000MS);

IF Timer.Q OR fbSend.Busy THEN
	Timer(IN:=FALSE);
	fbSend(SendString:= '$02Hello World ! $03',
			TXbuffer := TxBuffer, 
			Busy=> bSendBusy, 
			Error=> eSendErrorID);
END_IF

 fbReceive(	Prefix:= '$02',
			Suffix:= '$03',
			Timeout:= T#1S,
			ReceivedString:=sReceivedString,
			RXbuffer:= TxBuffer,
			StringReceived=> bStringReceived,
			Busy=> bReceiveBusy,
			Error=> eReceiveErrorID,
			RxTimeout=> bReceiveTimeout);
IF bStringReceived THEN
	nReceiveCounter := nReceiveCounter + 1 ;
	sLastReceiveString := sReceivedString;
END_IF

ClearComBuffer(Buffer:= TxBuffer);

END_FUNCTION_BLOCK

// ---- POUs/Testprogramme/Hintergrund_fasttask.TcPOU
PROGRAM Hintergrund_fasttask
VAR
	Waage1: WaageBufferKomunikation;
	Waage2: WaageBufferKomunikation;
	Waage3: WaageBufferKomunikation;
	Waage4: WaageBufferKomunikation;
END_VAR


Waage1(myWaage:= Waage_1, myTxBuffer:= TxBuffer1, myRxBuffer:= RxBuffer1, Waage => Waage_1);

Waage2(myWaage:= Waage_2, myTxBuffer:= TxBuffer2 , myRxBuffer:= RxBuffer2, Waage => Waage_2);

Waage3(myWaage:= Waage_3, myTxBuffer:= TxBuffer3 , myRxBuffer:= RxBuffer3, Waage => Waage_3);

Waage4(myWaage:= Waage_4, myTxBuffer:= TxBuffer4 , myRxBuffer:= RxBuffer4, Waage => Waage_4);

END_PROGRAM

// ---- POUs/Testprogramme/ModbusMasterApplication.TcPOU
(* 	Modbus-RTU Master
 * 	sample application
 *
 * 	Modbus master accessing up to 8 modbus slaves
 *)
PROGRAM ModbusMasterApplication
VAR
	MBKeyboard : ARRAY[1..16] OF WORD;	(* Keyboard area for a SAE-Stahl terminal e. g. MT-45 or MT-50 *)
	MBdata : ARRAY[0..99] OF WORD;		(* The size of this array can be adapted to the modbus slaves register area *)
	ModbusAddress : ARRAY[1..8] OF BYTE := [1,2,3,4,5,6,7,8]; (* list of Modbus slave addresses *)
	MB: ModbusRtuMaster_PcCOM;
	FtrigBusy: F_TRIG;
	timeoutvalue: TIME := T#300ms;		(* timeout while waiting for an answer of the modbus slave *)
	Unit: BYTE;
	state: INT;
	busy: BOOL;
	LastErrorstate: INT;
	LastModbusError: ST_ModbusErrorDiagnostics;
	CounterError: DINT;
	CounterSuccess: DINT;
	i: INT;
	x: INT;
END_VAR


CASE state OF
	0:
		MB.ReadRegs(Execute:= FALSE); (* initialize *)

		(* select one out of eight Modbus slaves *)
		Unit := Unit + 1;
		IF Unit > 8 THEN
			Unit := 1;
		END_IF

		state := state + 1;

	(*=================*)
	(* test data only!!! *)
		IF Unit = 1 THEN
	 		x := x + 1;
			IF x >= 100 THEN x := 0;
		END_IF
			FOR i := 0 TO 9 DO
				MBdata[i] := i*100 + x;
			END_FOR
		END_IF
	(*=================*)

	1:	(* Read Keyboard *)
		MB.ReadRegs(
			UnitID:= ModbusAddress[Unit], (* station address *)
			Quantity:= SIZEOF(MBKeyboard) / 2,	(* WORDs *)
			MBAddr:= 0,
			cbLength:= SIZEOF(MBKeyboard),
			pMemoryAddr:= ADR(MBKeyboard),
			Execute:= TRUE,
			Timeout:= timeoutvalue,
			Busy => busy	);
		IF NOT busy THEN
			MB.ReadRegs(Execute:= FALSE);
			IF MB.Error THEN
				state := 0;
			ELSE
				state := state + 1;
			END_IF
		END_IF

	2:	(* Read MBdata[20..40] from terminal address 100 *)
		MB.ReadRegs(
			UnitID:= ModbusAddress[Unit], (* station address *)
			Quantity:= 20,	(* WORDs *)
			MBAddr:= 100,
			cbLength:= 40,	(* 20 words *)
			pMemoryAddr:= ADR(MBdata[20]),
			Execute:= TRUE,
			Timeout:= timeoutvalue,
			Busy => busy	);
		IF NOT busy THEN
			MB.ReadRegs(Execute:= FALSE);
			state := state + 1;
		END_IF

	3:	(* Write value MBdata[0..9] to terminal registers 60-70 *)
		MB.WriteRegs(
			UnitID:= ModbusAddress[Unit], (* station address *)
			Quantity:= 10, (* WORDs *)
			MBAddr:= 60,
			cbLength:= SIZEOF(MBdata),	(* maximum buffer size *)
			pMemoryAddr:= ADR(MBdata[0]),
			Execute:= TRUE,
			Timeout:= timeoutvalue,
			Busy => busy	);
		IF NOT busy THEN
			MB.WriteRegs(Execute:= FALSE);
			state := 0;
		END_IF
END_CASE

FtrigBusy(CLK:=mb.BUSY );
IF FtrigBusy.Q THEN
	IF mb.Error THEN
		LastModbusError := mb.ErrorDiagnostics;
		LastErrorstate := state;
		CounterError := CounterError + 1;
	ELSE
		CounterSuccess := CounterSuccess + 1;
	END_IF
END_IF

END_PROGRAM
